(*
version 1.0	4 aug 2006
programmer 	hugo
tested by		tobias

this Function Block extracts the 8 Bits from a byte

executioin TIME on wago 750-841 = 13us
*)
B0 := IN.0;
B1 := IN.1;
B2 := IN.2;
B3 := IN.3;
B4 := IN.4;
B5 := IN.5;
B6 := IN.6;
B7 := IN.7;
END_FUNCTION_BLOCK

(* POU Engineering/signal processing/Byte_to_Range, ST *)
FUNCTION Byte_to_Range : REAL
VAR_INPUT
	X : BYTE;
	low : REAL;
	high : REAL;
END_VAR
VAR
END_VAR

(*
version 1.0	9. jan 2008
programmer 	hugo
tested by		tobias

Byte_to_Range converts a Byte into a real between low and high.

*)
Byte_to_Range := (high - low) * X / 255.0 + low;


(* revision history
hm	9. jan 2008		rev 1.0
	original version

*)
END_FUNCTION

(* POU String/BYTE_TO_STRH, ST *)
FUNCTION BYTE_TO_STRH : STRING
VAR_INPUT
	IN : BYTE;
END_VAR
VAR
	temp : BYTE;
	PT : POINTER TO BYTE;
END_VAR

(*
version 1.2	15 dec 2007
programmer 	hugo
tested by		tobias

BYTE_TO_STRINGH converts a Byte to a String of Hexadecimal represented by '0' .. '9' and 'A' .. 'F'.
The lowest order Character will be on the right and the high order Character on the left.

*)
(* read pointer to output string *)
PT := ADR(BYTE_TO_STRH);
(* calculate high order hex value *)
temp := SHR(in,4);
(* convert value to hex character *)
IF temp <= 9 THEN temp := temp + 48; ELSE temp := temp + 55; END_IF;
(* write friat character to output string *)
PT^ := temp;
(* calculate low order hex value *)
temp := in AND 2#00001111;
IF temp <= 9 THEN temp := temp + 48; ELSE temp := temp + 55; END_IF;
(* increment pointer and wirte low order character *)
pt := pt + 1;
pt^ := temp;
(* set pointer at the end of the output string and close the string with 0 *)
pt := pt + 1;
pt^:= 0;


(* code before rev 1.2
FOR i := 1 TO 2 DO
	X := in AND 2#1111;
	IF X <= 9 THEN X := X + 48; ELSE X := X + 55; END_IF;
	Cx := CHR(X);
	temp := CONCAT(Cx, temp);
	in := SHR(in,4);
END_FOR;
BYTE_TO_STRH := temp;
*)

(* revision history

hm		9.6.2007		rev 1.0		
	original version 

hm		11.9.2007		rev 1.1		
	changed coding for compatibility with twincat, under twincat concat cannot have a function as argument.	

hm		15 dec 2007		REV 1.2
	changed code for higher performance
*)
END_FUNCTION

(* POU Engineering/conversion/C_to_F, ST *)
FUNCTION C_to_F : REAL
VAR_INPUT
	celsius : REAL;
END_VAR
VAR
END_VAR

(*
version 1.0	4 aug 2006
programmer 	hugo
tested by		tobias

this function converts celsius  to fahrenheit 

*)
C_to_F := celsius * 1.8 + 32;
END_FUNCTION

(* POU Engineering/conversion/C_to_K, ST *)
FUNCTION C_to_K : REAL
VAR_INPUT
	Celsius : REAL;
END_VAR
VAR
END_VAR

(*
version 1.0	4 dec 2006
programmer 	hugo
tested by		tobias

this function converts celsius to kelvin
*)
C_to_K := Celsius - 273.15;
END_FUNCTION

(* POU Mathematical/Complex/CABS, ST *)
FUNCTION CABS : REAL
VAR_INPUT
	X : complex;
END_VAR
VAR
END_VAR

(*
version 1.0	21 feb 2008
programmer 	hugo
tested by	oscat

this function the aboslute value of a complex number

*)
CABS := HYPOT(x.re, x.im);


(* revision history
hm	21. feb 2008	rev 1.0
	original version

*)
END_FUNCTION

(* POU Engineering/measurements/Calibrate, ST *)
FUNCTION_BLOCK Calibrate
VAR_INPUT
	X : REAL;
	CO : BOOL;
	CS : BOOL;
END_VAR
VAR_INPUT CONSTANT
	Y_Offset : REAL;
	Y_Scale : REAL;
END_VAR
VAR_OUTPUT
	Y : REAL;
END_VAR
VAR RETAIN
	offset : REAL;
	Scale : REAL := 1;
END_VAR

(*
	version 1.2	22 feb 2007
	programmer 	hugo
	tested BY		hans

Calibrate allows for offset and scale calibration of an analog input.
offset is calibrated to a stored reference Y_offset while CO is true.
after the offset is calibrated, scale can be calibrated to a reference value Y_scale while CS is true.
*)
(* check for calibration *)
IF CO THEN
	Offset := Y_Offset - X;
ELSIF CS THEN
	scale := Y_scale / (X+Offset);
END_IF;
(* calculate output *)
Y := (X + Offset) * Scale;


(* revision history
hm 22.2.2007		rev 1.2
	changed VAR RETAIN PERSISTENT to VAR RETAIN for better compatibility
	wago lon contollers do not support persisitent

*)
END_FUNCTION_BLOCK

(* POU String/CAPITALIZE, ST *)
FUNCTION CAPITALIZE : STRING
VAR_INPUT
	str : STRING;
END_VAR
VAR
	PT : POINTER TO BYTE;
	pos : INT;
	L : INT;
	first : BOOL := TRUE;
END_VAR

(*
version 1.0	4. mar 2008
programmer 	hugo
tested by		tobias

uppercase returns str while all letters a..z and ä,ö,ü are converted to uppercase

*)
PT := ADR(CAPITALIZE);
CAPITALIZE := str;
L := LEN(str);
FOR pos := 1 TO l DO
	IF first THEN
		pt^ := TO_UPPER(pt^);
	END_IF;
	(* remember in first if the next char needs to capitalized *)
	IF pt^ = 32 THEN first := TRUE; ELSE first := FALSE; END_IF;
	PT := pt + 1;
END_FOR;

(* revision histroy
hm		4. mar 2008	rev 1.0
	original release

*)	
END_FUNCTION

(* POU String/TO_UPPER, ST *)
FUNCTION TO_UPPER : BYTE
VAR_INPUT
	IN : BYTE;
END_VAR
VAR
END_VAR

(*
version 1.0	6 mar 2008
programmer 	hugo
tested by		tobias

to_upper converts a character from lowercase to uppercase

*)
IF extended_ascii THEN
	IF ((in > 96) AND (in < 123)) OR ((in > 223) AND (in <> 247) AND (in <> 255)) THEN
		TO_UPPER := in AND 16#DF;
	ELSE
		TO_UPPER := in;
	END_IF;
ELSE
	IF ((in > 96) AND (in < 123)) THEN
		TO_UPPER := in AND 16#DF;
	ELSE
		TO_UPPER := in;
	END_IF;
END_IF;

(* revision history
hm		6. mar 2008	rev 1.0
	original version

*)
END_FUNCTION

(* POU Mathematical/Complex/CARG, ST *)
FUNCTION CARG : REAL
VAR_INPUT
	X : complex;
END_VAR
VAR
END_VAR

(*
version 1.0	21 feb 2008
programmer 	hugo
tested by	oscat

this function calculates the phase angle (argument) of a complex number

*)
CARG := ATAN(X.im / X.re);



(* revision history
hm	21. feb 2008	rev 1.0
	original version


*)
END_FUNCTION

(* POU Mathematical/Complex/CCON, ST *)
FUNCTION CCON : complex
VAR_INPUT
	X : complex;
END_VAR
VAR
END_VAR

(*
version 1.0	21 feb 2008
programmer 	hugo
tested by	oscat

this function calcucates the conjugation of a complex number

*)
CCON.re := x.re;
CCON.im := -x.im;


(* revision history
hm	21. feb 2008	rev 1.0
	original version

*)
END_FUNCTION

(* POU Logic/gate logic/check_parity, ST *)
FUNCTION check_parity : BOOL
VAR_INPUT
	in : DWORD;
	p : BOOL;
END_VAR
VAR
END_VAR

(*
version 1.3	18 feb 2008
programmer 	hugo
tested by		tobias

this function checks for an even partity for a dword and partity bit.

*)
check_parity := NOT p;
WHILE in > 0 DO
	check_parity := check_parity XOR in.0 XOR in.1 XOR in.2 XOR in.3;
	in := SHR(in,4);
END_WHILE;

(* code before rev 1.2
WHILE in > 0 DO
	IF in.0 THEN cnt := cnt + 1; END_IF;
	in := SHR(in,1);
END_WHILE;
check_parity := even(cnt) XOR P;
*)


(* revision history

rev 1.0 HM  1.oct.2006

rev 1.1 hm	10.sep.2007
	changed algorithm to improove performance

rev 1.2	hm	8 dec 2007
	changed algorithm to improove performance

rev 1.3 hm	18. feb 2008
	changed algorithm to improove performance
*)
END_FUNCTION

(* POU String/CHR, ST *)
FUNCTION CHR : STRING
VAR_INPUT
	C : BYTE;
END_VAR
VAR
	PT : POINTER TO BYTE;
END_VAR

(*
version 1.1	4. feb 2008
programmer 	hugo
tested by		tobias

CHR creates a character from a byte input and stuffs it in a one character length string.

*)
PT := ADR(CHR);
PT^ := C;
pt := pt + 1;
pt^ := 0;

(* revision history
hm		16 jan 2007		rev 1.0
	original version

hm		4. feb. 2008		rev 1.1
	return string would not be terminated properly
*)
END_FUNCTION

(* POU Mathematical/Geometry/circle_A, ST *)
FUNCTION circle_A : REAL
VAR_INPUT
	rx : REAL;
	ax : REAL;
END_VAR
VAR
END_VAR

(*
version 1.2	22. feb 2008
programmer 	hugo
tested by		tobias

circle_A calculates the Area of a circle segement if ax = 360 the whole circle is calculated


*)
circle_A := Rx * RX * 8.726646E-3 * Ax;

(* revision histroy
hm	16. oct 2007	rev 1.0
	original version

hm	4. dec 2007		rev 1.1
	changed code for better performance

hm	22. feb 2008	rev 1.2
	improved performance
*)
END_FUNCTION

(* POU Mathematical/Geometry/circle_C, ST *)
FUNCTION circle_C : REAL
VAR_INPUT
	Rx : REAL;
	Ax : REAL;
END_VAR
VAR
END_VAR

(*
version 1.1	22 feb 2008
programmer 	hugo
tested by		tobias

circle_C calculates the Circumference of a circle  if ax = 360 the whole circle is calculated

*)
circle_C := 1.7453293E-2 * Rx * Ax;

(* revision histroy
hm	16. oct 2007	rev 1.0
	original version

hm	22. feb 2008	rev 1.1
	improved performance
*)
END_FUNCTION

(* POU Building/electrical/click, ST *)
FUNCTION_BLOCK click
VAR_INPUT
	in : BOOL;
END_VAR
VAR_OUTPUT
	Q : BOOL;
	single : BOOL;
	double : BOOL;
	triple : BOOL;
	status: BYTE;
END_VAR
VAR_INPUT CONSTANT
	T_debounce : TIME := t#10ms;
	T_short : TIME := t#200ms;
	T_pause : TIME := t#500ms;
	T_reconfig : TIME := t#1m;
END_VAR
VAR
	debounce : TON;
	tx : TIME;
	last : TIME;
	init : BOOL;
	edge : BOOL;
	standby: BOOL;
	state: INT;
END_VAR

(*
version 1.2	15 sep 2007
programmer 	oscat
tested by		tobias

click checks an input for single, double or tripple click and sets the corresponding output single, doulbe or triple for the time the input stays high at the last click.
the maximum high and low time for a click can beconfigrured with setup variables.
the input cinfigures itself to be high or low active dependung on which state the input stays longer than t_reconfig.

*)
(* read system time *)
tx := DWORD_TO_TIME(T_PLC_MS());

(* set last and tx if never started before *)
IF NOT init THEN
	init := TRUE;
	last := tx;
	debounce.PT := T_debounce;
	standby := in;
END_IF;

(* debounce input *)
debounce(in := in XOR standby);
Q := debounce.Q;

(* delete outputs if input is inactive *)
IF NOT Q THEN
	single := FALSE;
	double := FALSE;
	triple := FALSE;
	status := 110;
END_IF;

(* check for input edge *)
IF Q XOR edge THEN
	edge := in;
	last := tx;
	IF Q THEN state := state + 1; END_IF;
END_IF;

IF (q AND tx - last >= T_short) OR (NOT q AND tx - last >= t_pause) THEN
	CASE state OF
		1:	single := TRUE;
			status := 111;
		2:	double := TRUE;
			status := 112;
		3:	triple := TRUE;
			status := 113;
	END_CASE;
	state := 0;
END_IF;

(* determine if high or low active *)
IF tx - last >= t_reconfig THEN
	standby := in;
	last := tx;
END_IF;



(* revision history

15 Feb 2007	rev 1.0	hm
	created original version

18.5.2007		rev 1.1 hm
	corrected an error while execution would stop after t_reconfig elapsed.

15.9.2007		rev 1.2 hm
	replaced Time() with T_PLC_MS for compatibility and performance reasons

*)
END_FUNCTION_BLOCK

(* POU Logic/generators/clk_div, ST *)
FUNCTION_BLOCK clk_div
VAR_INPUT
	clk : BOOL;
	rst: BOOL;
END_VAR
VAR_OUTPUT
	Q0 : BOOL := 0;
	Q1 : BOOL := 0;
	Q2 : BOOL := 0;
	Q3 : BOOL := 0;
	Q4 : BOOL := 0;
	Q5 : BOOL := 0;
	Q6 : BOOL := 0;
	Q7 : BOOL := 0;
END_VAR
VAR
	cnt: BYTE := 0;
END_VAR

(*
version 1.1	2 jan 2008
programmer 	hugo
tested by		tobias

this is a clock divider
each output divides the signal by 2
Q0 = clk / 2 , Q1 = Q0 / 2 and so on.
the outputs have a 50% duty cycle each.


*)
IF rst THEN
	cnt:= 0;
	Q0 := 0;
	Q1 := 0;
	Q2 := 0;
	Q3 := 0;
	Q4 := 0;
	Q5 := 0;
	Q6 := 0;
	Q7 := 0;
ELSIF clk THEN
	cnt:= cnt +1;
	Q0 := cnt.0;
	Q1 := cnt.1;
	Q2 := cnt.2;
	Q3 := cnt.3;
	Q4 := cnt.4;
	Q5 := cnt.5;
	Q6 := cnt.6;
	Q7 := cnt.7;
END_IF;

(* revision history
hm	4. aug. 2006	rev 1.0
	original version

hm	2. jan 2008		rev 1.1
	improved performance

*)
END_FUNCTION_BLOCK

(* POU Logic/generators/CLK_N, ST *)
FUNCTION_BLOCK CLK_N
VAR_INPUT
	N : INT;
END_VAR
VAR_OUTPUT
	Q : BOOL;
END_VAR
VAR
	edge : BOOL := 0;
	stime: DWORD;
	clk: BOOL;
END_VAR

(*
version 1.0	17 sep 2007
programmer 	hugo
tested by		tobias

clk_N uses the internal sps time to generate one pulse every N ms
every pulse is only valid for one cycle so that a edge trigger is not necessary
clk_N generates pulses depending on the accuracy of the system clock.
The input N controlls the period time of the clock.
N=0 equals 1ms, N=1 equals 2ms, N=2 equals 4ms, N=3 equals 8ms ....

be careful, 1ms clocks will only work on very powerful sps cpu's
*)
stime := SHR(T_PLC_MS(),N);
clk := stime.0;
Q := clk XOR edge;
edge := CLK;

(* revision history
hm	16. dec 2007		rev 1.0
	original version

*)
END_FUNCTION_BLOCK

(* POU XTEST/Ideas/stime, ST *)
FUNCTION_BLOCK stime
VAR_INPUT
END_VAR
VAR_OUTPUT
	tx : DWORD;
END_VAR
VAR
	last_time: DWORD;
	bit31: BOOL;
END_VAR

(* this function block makes sure that the timer of a siemens sps counts from 0 - 2^32-1. *)
(* this FB is only necessary for siemens sps
the siemens sps timer counts from 0 to 2^31-1 and starts at 0 sfter overrun.
this means that the bit 31 (the highest bit ) will never be used and therefore
a problem arises when t2 - t1 is checked.
t2 - t1 is always valid also in an timer overrun situation where the time t1 is very high and t2 is very low.
the result of the subtraction t2 - t1 however is still valid.
this calculation does not work for siemens because the highest bit is not used.

this module stores the highest bit, changes the highest bit at every overrun occurence and stuffs ther highest bit in the output.
the output is then used by t_plc_us and t_plc_ms.

the correction needs and fb and not a function because the value of the highest bit has to be stored.

do never use this function block in a codesys environment. the timer in codesys is correct and runs from 0 to 2^32-1
*)

(* read the system timer *)
tx := TIME_TO_DWORD(TIME());

(* check for overrun *)
IF tx < last_time THEN
	(* an overrun has occured, change the value of the highest bit *)
	bit31 := NOT bit31;
END_IF;

(* remember the last system time for the next overrun check *)
last_time := tx;

(* stuff the highest bit into the timer value *)
tx.31 := bit31;
END_FUNCTION_BLOCK

(* POU Logic/generators/CLK_Prg, ST *)
	FUNCTION_BLOCK CLK_Prg
VAR_INPUT
	PT : TIME := t#10ms;
END_VAR
VAR_OUTPUT
	Q : BOOL := 0;
END_VAR
VAR
	init : BOOL := FALSE;
	last : TIME;
	tx: TIME;
END_VAR

(*
version 1.2	17 sep 2007
programmer 	hugo
tested by		tobias

clk_prg uses the internal sps time to generate a clock with programmable period time.
the period time is defined for 10ms .. 65s
the first cycle after start is a clk pulse and then depending on the programmed period time a delay.
every pulse is only valid for one cycle.
the accuracy of clk_prg is depending on the accuracy of the system clock.

*)
(* read system time *)
tx := DWORD_TO_TIME(T_PLC_MS());

(* initialize on startup *)
IF NOT init THEN
	init := TRUE;
	last := tx - pt;
END_IF;

(* generate output pulse when next_pulse is reached *)
IF tx - last >= pt THEN
	Q := TRUE;
	last := tx;
ELSE
	Q := FALSE;
END_IF;


(* revision hiostory

hm 25 feb 2007	rev 1.1
	rewritten code for higher performance
	pt can now be changed during runtime

hm	17. sep 2007	rev 1.2
	replaced time() with t_plc_ms() for compatibility reasons

*)
END_FUNCTION_BLOCK

(* POU Logic/generators/CLK_Pulse, ST *)
FUNCTION_BLOCK CLK_Pulse
VAR_INPUT
	PT : TIME := t#10ms;
	N : INT := 0;
	rst : BOOL := 0;
END_VAR
VAR_OUTPUT
	Q : BOOL := 0;
	cnt : INT := 0;
	run : BOOL := 0;
END_VAR
VAR
	pti : TIME := t#0ms;
	next_pulse: TIME := T#0s;
	overflow: BOOL := FALSE;
	tx: TIME;
END_VAR

(*
version 1.1	17 sep 2007
programmer 	hugo
tested by		tobias

clk_pulse uses the internal sps time to generate a clock with programmable period time.
the period time is defined for 10ms .. 65s.
pulse generation is continuous if N = 0 and for n pulses otherwise.
if the period time is set to less then 10ms the min clock perid is 10ms.
the first cycle after start is a clk pulse and then depending on the programmed period time a delay.
every pulse is only valid for one cycle so that a edge trigger is not necessary
clk_prg depending on the accuracy of the system clock.

*)
(* read system *)
tx := DWORD_TO_TIME(T_PLC_MS());


IF rst THEN
	run := FALSE;
	pti := t#0ms;
	next_pulse := t#0ms;
	overflow := FALSE;
	Q := FALSE;
	cnt := 0;
ELSIF cnt <= N OR N = 0 THEN
	IF NOT run THEN
		next_pulse := tx;
		run := TRUE;
		IF pt < T#10ms THEN PTI := T#10ms; ELSE pti := pt; END_IF;
	END_IF;
	IF tx >= next_pulse AND NOT overflow AND (cnt < N OR N = 0) THEN
		Q := TRUE;
		cnt := cnt + 1;
		IF next_pulse + pti < next_pulse THEN
			overflow := TRUE;
		END_IF;
		next_pulse := next_pulse + pti;
	ELSE
		Q := FALSE;
		IF cnt = N THEN run := FALSE; END_IF
		IF tx <= next_pulse THEN overflow := FALSE; END_IF;
	END_IF;
END_IF

(* revision history
hm		4. aug 2006		rev 1.0
	original version

hm		17. sep 2007	rev 1.1
	replaced time() with T_PLC_S() fr compatblity reasons

*)
END_FUNCTION_BLOCK

(* POU Mathematical/Geometry/cone_V, ST *)
FUNCTION cone_V : REAL
VAR_INPUT
	rx : REAL;
	hx : REAL;
END_VAR
VAR
END_VAR

(*
version 1.1	4 dec 2007
programmer 	hugo
tested by		tobias

cone_V calculates the Volume of a cone

*)
cone_V := 1.047197551 * RX * RX * hx;

(* revision histroy
hm	17. oct 2007	rev 1.0
	original version

hm	4. dec 2007		rev 1.1
	changed code for better performance

hm	22. feb 2008	rev 1.2
	changed code for better performance
*)
END_FUNCTION

(* POU Engineering/control/control_set1, ST *)
FUNCTION_BLOCK control_set1
VAR_INPUT
	Kt : REAL;
	Tt : REAL;
	PI : BOOL;
	PID : BOOL;
END_VAR
VAR_INPUT CONSTANT
	P_K : REAL := 0.5;
	PI_K : REAL := 0.45;
	PI_TN : REAL := 0.83;
	PID_K : REAL := 0.6;
	PID_TN : REAL := 0.5;
	PID_TV : REAL := 0.125;
END_VAR
VAR_OUTPUT
	KP : REAL;
	TN : REAL;
	TV : REAL;
	KI : REAL;
	KD : REAL;
END_VAR
VAR
END_VAR

(*
version 1.0	4 nov 2007
programmer 	hugo
tested by	tobias

takahashi calculates controller parameters for P, PI and PID controllers based on the ziegler nichols method.

*)
IF pi AND PID THEN
	KP := 0;
	TN := 0;
	TV := 0;
ELSIF PID THEN
	KP := PID_K * Kt;
	TN := PID_TN * Tt;
	TV := PID_TV * Tt;
ELSIF PI THEN
	KP := PI_K * Kt;
	TN := PI_TN * Tt;
ELSE
	KP := P_K * Kt;
END_IF;

(* KI and KD are calculated *)
IF tn > 0 THEN KI := KP / TN; ELSE KI := 0; END_IF;
KD := KP * TV;

(* revision history
hm	4. nov 2007		rev 1.0
	original version

*)
END_FUNCTION_BLOCK

(* POU Engineering/control/control_set2, ST *)
FUNCTION_BLOCK control_set2
VAR_INPUT
	KS : REAL;
	TU : REAL;
	TG : REAL;
	PI : BOOL;
	PID : BOOL;
END_VAR
VAR_INPUT CONSTANT
	P_K : REAL := 1.0;
	PI_K : REAL := 0.9;
	PI_TN : REAL := 3.33;
	PID_K : REAL := 1.2;
	PID_TN : REAL := 2;
	PID_TV : REAL := 0.5;
END_VAR
VAR_OUTPUT
	KP : REAL;
	TN : REAL;
	TV : REAL;
	KI : REAL;
	KD : REAL;
END_VAR
VAR
	TX : REAL;
END_VAR

(*
version 1.0	4 nov 2007
programmer 	hugo
tested by	tobias

takahashi calculates controller parameters for P, PI and PID controllers based on the ziegler nichols method.

*)
IF TU > 0 AND KS > 0 THEN TX := TG/TU/KS; END_IF;
IF pi AND PID THEN
	KP := 0;
	TN := 0;
	TV := 0;
ELSIF PID THEN
	KP := PID_K * TX;
	TN := PID_TN * TU;
	TV := PID_TV * TU;
ELSIF PI THEN
	KP := PI_K * TX;
	TN := PI_TN * TU;
ELSE
	KP := P_K * TX;
END_IF;

(* KI and KD are calculated *)
IF TN > 0 THEN KI := KP / TN; ELSE KI := 0; END_IF;
KD := KP * TV;

(* revision history
hm	4. nov 2007		rev 1.0
	original version

*)
END_FUNCTION_BLOCK

(* POU Logic/FF edge triggered/COUNT_BR, ST *)
FUNCTION_BLOCK COUNT_BR
VAR_INPUT
	SET : BOOL;
	IN : BYTE;
	UP : BOOL;
	DN : BOOL;
	STEP : BYTE := 1;
	MX : BYTE := 255;
	RST : BOOL;
END_VAR
VAR_INPUT CONSTANT

END_VAR
VAR_OUTPUT
	CNT : BYTE;
END_VAR
VAR
	last_up: BOOL;
	last_dn: BOOL;
END_VAR

(*
	version 1.0	16 jan 2008
	programmer 	hugo
	tested BY	tobias

Count_R is a byte counter with independen up and dn inputs. the counter counts from 0 to mx and continues at 0 after is has reached mx
a step input sets the counters stepping width.

*)
IF rst THEN
	cnt := 0;
ELSIF set THEN
	cnt := LIMIT(0,in,mx);
ELSIF up AND NOT last_up THEN
	cnt := INT_TO_BYTE(inc(cnt,step,mx));
ELSIF dn AND NOT last_dn THEN
	cnt := INT_TO_BYTE(inc(cnt,-step,mx));
END_IF;
last_up := up;
last_dn := dn;

(* revision history
hm	16. jan 2008	rev 1.0
	original version

*)
END_FUNCTION_BLOCK

(* POU String/COUNT_CHAR, ST *)
FUNCTION COUNT_CHAR : INT
VAR_INPUT
	str : STRING;
	chr : BYTE;
END_VAR
VAR
	l: INT;
	pt : POINTER TO BYTE;
	pos: INT;
END_VAR


(*
version 1.0	29. feb 2008
programmer 		kurt
tested by		hugo

COUNT_CHAR how often a character CHAR occurs within a string STR.

*)
PT := ADR(str);
l := LEN(str);
COUNT_CHAR := 0;
FOR pos := 1 TO l DO
	IF pt^ = CHR THEN COUNT_CHAR := COUNT_CHAR + 1; END_IF;
    PT := PT + 1;
END_FOR;


(* revision history
hm		29. feb 2008	rev 1.0
	original version

*)
END_FUNCTION

(* POU Mathematical/Complex/CPOL, ST *)
FUNCTION CPOL : complex
VAR_INPUT
	L : REAL;
	A : REAL;
END_VAR
VAR
END_VAR

(*
version 1.0	21 feb 2008
programmer 	hugo
tested by	oscat

this function creates a complex numbers for the polar form with the inputs L (length) an A for Angle.

*)
CPOL.re := L * COS(A);
CPOL.im := L * SIN(A);


(* revision history
hm	21. feb 2008	rev 1.0
	original version

*)
END_FUNCTION

(* POU Logic/Others/CRC_CHECK, ST *)
FUNCTION CRC_CHECK : BOOL
VAR_INPUT
	pt : POINTER TO ARRAY[0..32000] OF BYTE;
	size : INT;
END_VAR
VAR_INPUT CONSTANT
	Polynom_L : DWORD;
	Polynom_32 : BOOL;
END_VAR
VAR
	temp: DWORD;
END_VAR

(*
version 1.0	9 jun 2007
programmer 	hugo
tested by		tobias

CRC_CHECK checks a block of data for a crc checksum and returns true is the checksum is 0 and therfore a error free data transmission.
the CRC Polynom is specified with the config variable Polynom_L which holds the lowest 32 bits of the polynom and Polynom_33 which holds bit 33 of the Polynom.
A Polynom x4 + X + 1 is represented by 10011.
The input data is an array of byte of any size, the function is called by CRC_CHECK(ADR(array),SIZEOF(array)).

*)
temp := CRC_GEN(pt, size, polynom_L, polynom_32, 0, 0, FALSE, FALSE);
IF temp = 0 THEN CRC_CHECK := TRUE; ELSE CRC_CHECK := FALSE; END_IF;

(* typical crc polynoms

CRC-4-ITU 			x4 + x + 1 					(ITU G.704, p. 12) 	0x3 or 0xC (0x9)
CRC-5-ITU 			x5 + x4 + x2 + 1 			(ITU G.704, p. 9) 	0x15 or 0x15 (0x0B)
CRC-5-USB 			x5 + x2 + 1 				(use: USB token packets) 	0x05 or 0x14 (0x9)
CRC-6-ITU 			x6 + x + 1 					(ITU G.704, p. 3) 	0x03 or 0x30 (0x21)
CRC-7 				x7 + x3 + 1 				(use: telecom systems, MMC) 	0x09 or 0x48 (0x11)
CRC-8-ATM 			x8 + x2 + x + 1 				(use: ATM HEC) 	0x07 or 0xE0 (0xC1)
CRC-8-CCITT 		x8 + x7 + x3 + x2 + 1 		(use: 1-Wire bus) 	0x8D or 0xB1 (0x63)
CRC-8-Dallas/Maxim 	x8 + x5 + x4 + 1 			(use: 1-Wire bus) 	0x31 or 0x8C (0x19)
CRC-8 				x8 + x7 + x6 + x4 + x2 + 1 	0xD5 or 0xAB (0x57)
CRC-8-SAE J1850 	x8 + x4 + x3 + x2 + 1 		0x1D or 0xB8
CRC-10 				x10 + x9 + x5 + x4 + x + 1 	0x233 or 0x331 (0x263)
CRC-12 				x12 + x11 + x3 + x2 + x + 1 (use: telecom systems) 	0x80F or 0xF01 (0xE03)
CRC-15-CAN 			x15 + x14 + x10 + x8 + x7 + x4 + x3 + 1 	0x4599 or 0x4CD1 (0x19A3)
CRC-16-Fletcher 	Not a CRC; see Fletcher's checksum 	Used in Adler-32 A & B CRCs
CRC-16-CCITT 	x16 + x12 + x5 + 1 (XMODEM,X.25, V.41, Bluetooth, PPP, IrDA; known as "CRC-CCITT") 	0x1021 or 0x8408 (0x0811)
CRC-16-IBM 	x16 + x15 + x2 + 1 (USB, many others; also known as "CRC-16") 	0x8005 or 0xA001 (0x4003)
CRC-24-Radix-64 	x24 + x23 + x18 + x17 + x14 + x11 + x10 + x7 + x6 + x5 + x4 + x3 + x + 1 	0x864CFB or 0xDF3261 (0xBE64C3)
CRC-32-Adler 	Not a CRC; see Adler-32 	See Adler-32
CRC-32-MPEG2 	x32 + x26 + x23 + x22 + x16 + x12 + x11 + x10 + x8 + x7 + x5 + x4 + x2 + x + 1 	0x04C11DB7 or 0xEDB88320 (0xDB710641) Also used in IEEE 802.3
CRC-32-IEEE 802.3 	x32 + x26 + x23 + x22 + x16 + x12 + x11 + x10 + x8 + x7 + x5 + x4 + x2 + x + 1 (V.42) 	0x04C11DB7 or 0xEDB88320 (0xDB710641)
CRC-32C (Castagnoli) 	x32 + x28 + x27 + x26 + x25 + x23 + x22 + x20 + x19 + x18 + x14 + x13 + x11 + x10 + x9 + x8 + x6 + 1 	0x1EDC6F41 or 0x82F63B78 (0x05EC76F1)
CRC-64-ISO 	x64 + x4 + x3 + x + 1 (use: ISO 3309) 	0x000000000000001B or 0xD800000000000000 (0xB000000000000001)
CRC-64-ECMA-182 	x64 + x62 + x57 + x55 + x54 + x53 + x52 + x47 + x46 + x45 + x40 + x39 + x38 + x37 + x35 + x33 + x32 + x31 + x29 + x27 + x24 + x23 + x22 + x21 + x19 + x17 + x13 + x12 + x10 + x9 + x7 + x4 + x + 1
(as described in ECMA-182 p.63) 	0x42F0E1EBA9EA3693 or 0xC96C5795D7870F42 (0x92D8AF2BAF0E1E85)

*)

(* revision history

hm		9.6.2007	rev 1.0		original version 

*)
END_FUNCTION

(* POU Logic/generators/D_Trig, ST *)
FUNCTION_BLOCK D_Trig
VAR_INPUT
	in : DWORD;
END_VAR
VAR_OUTPUT
	Q : BOOL;
	X : DWORD;
END_VAR
VAR
	last_in : DWORD;
END_VAR

(*
version 1.1	19. feb 2008
programmer 	hugo
tested by		tobias

this block is similar to the IEC Standard R_trig and F_trig but it monitors a DWORD, WORD or Byte Variable instead and generated an Output Pulse for one cycle only when the input has changed.
an additional output x (Dword) will state the chage of the input.
Example: the input has chaged from 0001 to 0010 then the output x will be 2.

*)
Q := in <> last_in;
X := in - last_in;
last_in := in;


(* revision history

hm 	4.09.2007		rev 1.0
	original version released

hm	19. feb. 2008	rev 1.1
	performance improvement
*)
END_FUNCTION_BLOCK

(* POU XTEST/Baustein Tests/date_test, ST *)
FUNCTION_BLOCK date_test
VAR_INPUT
END_VAR
VAR_OUTPUT
	fail : STRING;
	error : BOOL := FALSE;
	jahr : INT;
END_VAR
VAR
	i: INT;
	test : DATE;
	jan1 : DATE;
	dez31 : DATE;
END_VAR
IF error THEN RETURN; END_IF;

FOR i := 1970 TO 2099 DO
	jan1 := set_Date(i,1,1);
	dez31 := set_Date(i,12,31);

	(* test der funktion year_begin *)
	test := year_begin(i);
	IF test <> jan1 THEN
		error := TRUE;
		jahr := i;
		FAIL := 'year_begin';
	END_IF;

	(* test year *)
	IF year(jan1) <> i OR year(dez31) <> i THEN
		error := TRUE;
		jahr := i;
		fail := 'year';
	END_IF;
END_FOR;
END_FUNCTION_BLOCK

(* POU Time&Date/day_of_date, ST *)
FUNCTION day_of_date : INT
VAR_INPUT
	idate : DATE;
END_VAR
VAR
END_VAR


(*
	version 1.1	1 okt 2007
	programmer 	oscat
	tested BY		oscat

DAY_OF_DATE returns the days since 1.1.1970

*)
IF STEP7 THEN
	(* adjust step7 day by 7305 days because step7 date fornat starts at 1.1.1990  *)
	day_of_date := DWORD_TO_INT(DATE_TO_DWORD(idate) / 86400) + 7305;
ELSE
	day_of_date := DWORD_TO_INT(DATE_TO_DWORD(idate) / 86400);
END_IF;


(* revision history
hm		16.9.2007		rev 1.0
	original version

hm		1. okt 2007		rev 1.1
	added step7 compatibility

*)
END_FUNCTION

(* POU Time&Date/day_to_time, ST *)
FUNCTION day_to_time : TIME
VAR_INPUT
	input : REAL;
END_VAR
VAR
END_VAR

(*
version 1.0	4 aug 2006
programmer 	hugo
tested by		tobias

converts an amount of days in real to time 
*)
day_to_time := DWORD_TO_TIME(REAL_TO_DWORD(input * 86400000));
END_FUNCTION

(* POU Time&Date/days_delta, ST *)
FUNCTION days_delta : INT
VAR_INPUT
	date_1 : DATE;
	date_2 : DATE;
END_VAR
VAR
END_VAR

(*
version 1.1	27 dec 2006
programmer 	hugo
tested by		tobias

days_delta calculates the days between two dates. the days are calculated date_2 - date_1.

*)
days_delta := day_of_date(date_2) - day_of_date(date_1);

(* revision history
hm	27. dec 2006	rev 1.0
	original version

hm	16.9.2007		rev 1.1
	coorected an error in formula and changed algorithm to show positive and negative delta

*)
END_FUNCTION

(* POU Time&Date/DCF77, ST *)
FUNCTION_BLOCK DCF77
VAR_INPUT
	rec : BOOL;
	sdt : DT;
END_VAR
VAR_INPUT CONSTANT
	sync_timeout : TIME := t#2m;
	time_offset : INT := 1;
	dst_en : BOOL := TRUE;
END_VAR
VAR_OUTPUT
	TP : BOOL;
	DST : BOOL;
	weekday : INT;
	error: BOOL := TRUE;
	RTC : DT;
	RTC1 : DT;
	msec : INT;
	sync : BOOL;
END_VAR
VAR
	MEZ : DT;
	UTC : DT;
	state : INT;
	edge: BOOL;
	tx : TIME;
	ty: TIME;
	last : TIME;
	bits : ARRAY[0..58] OF BOOL;
	cnt : INT;
	i : INT;
	old_time : DT;
	minute : INT;
	hour : INT;
	day : INT;
	month : INT;
	year : INT;
	last_sync: TIME;
	t1: TIME;
	tz: TIME;
	init: BOOL;
END_VAR


(*
version 1.7	23. jan 2008
programmer 	hugo
tested by		tobias

this is a decoder for a DCF77 signal.
the decoder decodes the DCF77 signal and checks for a valid Date_Time.
since the dcf77 signal is only secured with a simple parity the decoder waits for two consecutive valid transmissions before it sets the output signals.
given a valid reception by the receiver the decoder can take up to 3 minutes to start its clocks the first time.
after a valid signal is detected the error output goes low and dignals a valid dcf signal from the receiver.
a tp is only valid for one program cycle to allow for external rtc setting.
after a valid signal is detected two independent internal clocks are started (RTC and RTC1), the seconds  of these clocks are generated by software since the dcf signal is only valid for minutes.
rtc is always utc ( world time) and rtc1 can be set to any time zone by setting the time_zone_offset and enabling dst for automatic summertime.
a sync output signals the the rtc and rtc1 are in sync with the dcf77 signal, if the dcf77 signal is lost for more then the sync time the sync output goes low
but the rtc and rtc1 outputs keep running based on software timing until a valid dcf77 signal is received again and triggers the clock.
in addition a millisecond output gives further resolutionof the clocks.
a dst output shows if daylight saving time is enables and the weekday output shows which day of week currently is ( 1= monday ... 7= sunday).


*)
(* if tp was set it should only be active for 1 cycle *)
TP := FALSE;

(* read system time *)
t1 := DWORD_TO_TIME(T_PLC_MS());
tx := t1 - last;

IF rec XOR edge THEN
	edge := rec;
	IF NOT rec AND tx > t#1700ms AND tx < t#2000ms THEN
		(* start condition reached *)
		state := 0;
		tp := NOT error;
	ELSIF NOT rec AND tx > t#700ms AND tx < t#1000ms THEN
		(* second switch detected *)
		IF state < 58 THEN state := state +1; ELSE state := 0; END_IF;
	ELSIF rec AND tx  < t#120ms THEN
		(* bit 0 detected  *)
		bits[state] := 0;
	ELSIF rec AND tx > t#120ms AND tx < t#250ms THEN
		(* bit 1 detected *)
		bits[state] := 1;
	ELSE
		(* error condition received signal is not valid *)
		error := TRUE;
		state := 0;
	END_IF;
	last := last + tx;
	IF rec AND state = 58 THEN
		error := FALSE;

		(* decode the bits and check for possible errors *)
		IF bits[0] OR NOT (bits[17] XOR bits[18]) OR NOT bits[20] THEN error := TRUE; END_IF;
		(* decode minute *)
		minute := 0;
		minute.0 := bits[21];
		minute.1 := bits[22];
		minute.2 := bits[23];
		minute.3 := bits[24];
		IF bits[25] THEN minute := minute + 10; END_IF;
		IF bits[26] THEN minute := minute + 20; END_IF;
		IF bits[27] THEN minute := minute + 40; END_IF;
		IF minute > 59 OR (bits[21] XOR bits[22] XOR bits[23] XOR bits[24] XOR bits[25] XOR bits[26] XOR bits[27] XOR bits[28]) THEN error := TRUE; END_IF;

		(* decode hour *)
		hour := 0;
		hour.0 := bits[29];
		hour.1 := bits[30];
		hour.2 := bits[31];
		hour.3 := bits[32];
		IF bits[33] THEN hour := hour + 10; END_IF;
		IF bits[34] THEN hour := hour +20; END_IF;
		IF hour > 23 OR (bits[29] XOR bits[30] XOR bits[31] XOR bits[32] XOR bits[33] XOR bits[34] XOR bits[35]) THEN error := TRUE; END_IF;

		(* decode day of month *)
		day := 0;
		day.0 := bits[36];
		day.1 := bits[37];
		day.2 := bits[38];
		day.3 := bits[39];
		IF bits[40] THEN day := day + 10; END_IF;
		IF bits[41] THEN day := day + 20; END_IF;
		IF day > 31 THEN error := TRUE; END_IF;

		(* decode day of week *)
		weekday := 0;
		weekday.0 := bits[42];
		weekday.1 := bits[43];
		weekday.2 := bits[44];
		IF weekday > 7 OR weekday < 1 THEN error := TRUE; END_IF;

		(* decode month *)
		month := 0;
		month.0 := bits[45];
		month.1 := bits[46];
		month.2 := bits[47];
		month.3 := bits[48];
		IF bits[49] THEN month := month +10; END_IF;
		IF month > 12 THEN error := TRUE; END_IF;

		(* decode year *)
		year := 0;
		year.0 := bits[50];
		year.1 := bits[51];
		year.2 := bits[52];
		year.3 := bits[53];
		IF bits[54] THEN year := year + 10; END_IF;
		IF bits[55] THEN year := year + 20; END_IF;
		IF bits[56] THEN year := year + 40; END_IF;
		IF bits[57] THEN year := year + 80; END_IF;

		(* check parity for bits 36 to 58 *)
		cnt := 0;
		FOR i := 36 TO 58 DO IF bits[i] THEN cnt := cnt + 1; END_IF; END_FOR;
		IF NOT even(cnt) THEN error := TRUE; END_IF;

		(* time must be valid for two cycles to clear error flag *)
		IF NOT error THEN
			(* set outputs *)
			old_time := mez;
			IF year >= 70 THEN year := year + 1900; ELSE year := year + 2000; END_IF;
			mez := set_DT(year,month,day,hour,minute,0);
			DST := bits[17];
			IF DST THEN
				UTC := DWORD_TO_DT(DT_TO_DWORD(mez) - 7200);
			ELSE
				UTC := DWORD_TO_DT(DT_TO_DWORD(mez) - 3600);
			END_IF

			(* set trigger signal only if the receiver has received 2 successive minutes *)
			IF mez <> old_time + t#1m THEN error := TRUE ; END_IF;
		END_IF;
	END_IF;
END_IF;

(* this portion implements a free running clock which is triggered by the dcf77 signal *)
tz := DWORD_TO_TIME(INT_TO_DWORD(ABS(time_offset))* 3600000);

(* input sdt is copied to utc at first power up *)
IF NOT init THEN
	init := TRUE;
	utc := sdt;
	tp := TRUE;
END_IF;

IF tp THEN
	rtc := utc;
	IF DST AND dst_en THEN
		IF time_offset < 0 THEN	rtc1 := rtc - tz + t#1h; ELSE rtc1 := rtc + tz + t#1h; END_IF;
	ELSE
		IF time_offset < 0 THEN rtc1 := rtc - tz; ELSE rtc1 := rtc + tz; END_IF;
	END_IF;
	sync := TRUE;
	last_sync := last;
	ty := last;
ELSIF rtc > DWORD_TO_DT(0) AND T1 - ty >= t#1s THEN
	rtc := rtc + t#1s;
	rtc1 := rtc1 + t#1s;
	ty := ty + t#1s;
	sync := ty - last_sync < sync_timeout AND last_sync > DWORD_TO_TIME(0);
	weekday := weekday(DT_TO_DATE(rtc1));
	DST := dst_en AND DST(utc);
END_IF;
msec := TIME_TO_INT(t1 - ty);



(* decode information
bits		content
0			Bitwert immer 0
1 bis 14	reserviert für Betriebsinformationen (nicht für DCF77-Nutzer bestimmt)
15			Rufbit für Alarmierung der PTB-Mitarbeiter
			(bis Mai 2003: Bitwert = 0 falls normale Antenne in Verwendung; 1 = Backupantenne)
16			Bitwert = 1 falls ein Wechsel von MEZ nach MESZ oder umgekehrt bevorsteht; Dauer der Anzeige: 1 Stunde
17 + 18	gültige Zeit = MEZ, falls Bit 17=0 und Bit 18=1
			gültige Zeit = MESZ, falls Bit 17=1 und Bit 18=0
19			Bitwert = 1 falls innerhalb den nächsten 59 Minuten eine Schaltsekunde angeordnet ist. Beim Einfügen einer Schaltsekunde wird anstelle der 59. die 60. Sekundenmarke weggelassen und in der 58. erfolgt ausnahmsweise ein Trägerabfall.
20			Startbit für Zeitinformation (immer 1)
21 - 27		1, 2, 4, 8, 10, 20, 40 Minuten (bitweise Addition)
28			Prüfbit (gerade Parität) für die Bits 21-27
29 - 34		1, 2, 4, 8, 10, 20 Stunden (bitweise Addition)
35			Prüfbit (gerade Parität) für die Bits 29-34
36 - 41		Tagesnummer im aktuellen Monat: 1, 2, 4, 8, 10, 20 (bitweise Addition)
42 - 44		Tagesnummer in der aktuellen Woche: 1, 2, 4 (bitweise Addition)
45 - 49		Monatsnummer: 1, 2, 4, 8, 10 (bitweise Addition)
50 - 57		Jahr (zweistellig): 1, 2, 4, 8, 10, 20, 40, 80 (bitweise Addition)
58			Prüfbit (gerade Parität) füR die Bits 36-57

*)
(* revision history

hm 2.feb 2007		rev 1.1
	change wday and dst outputs when there is no dcf reception

hm	26.feb 2007		rev 1.2
	changed statements where t#1h would be substracted from DT.
	under certain conditions the compiler would crash translating this statement

hm	17. sep 2007	rev 1.3
	replaced time() with T_PLC_MS() for compatibility reasons

hm	24. oct 2007	rev 1.4
	changed dst calculation because function dst was upgraded no error in DCF77 only a change in DST

hm	12. nov 2007	rev 1.5
	changed time_offset from time to integer to allow for negative offset time zones

hm	8. dec 2007		rev 1.6
	corrected an error in time_zone calculation

hm 23. jan 2008		rev 1.7
	added sdt input which is used to initialize rtc and rtc1 during first cycle. 
*)
END_FUNCTION_BLOCK

(* POU Time&Date/DST, ST *)
FUNCTION DST : BOOL
VAR_INPUT
	utc : DT;
END_VAR
VAR
	yr : INT;
	yr4 : DWORD;
	ltc: DWORD;
	idate : DWORD;
END_VAR

(*
version 1.2	1 dec 2007
programmer 	hugo
tested by		tobias

this functions returns TRUE IF dst TIME is active 
the FUNCTION calculates automatically for any year betweek 1970 AND 2099 
wheather daylight savings is on OR off 
the summertime calculation is done according to european standards.
dst will become TRUE AT 01:00 utc in the morning FOR the respective days 
AND it will become FALSE after daylight savings TIME is switched back end OF october at 01:00 utc

*)
yr := year(DT_TO_DATE(utc));
ltc := DT_TO_DWORD(utc);
idate := DT_TO_DWORD(set_DT(yr,3,31,1,0,0));
yr4 := SHR(5*yr,2);
IF idate - ((yr4+4) MOD 7)*86400 <= ltc AND idate + (214 - (yr4+1) MOD 7)*86400 > ltc THEN DST := TRUE; ELSE DST := FALSE; END_IF;

(* revision history
hm	4. aug 2006		rev 1.0
	original version

hm	24. okt 2007	rev 1.1
	deleted time_zone_offset input because dst is generally at 01:00 utc and not mesz
	uk starts 01:00 utc and also greece

hm	1. dec 2007		rev 1.2
	changed code to improove performance

*)

(*
Equation used TO calculate the beginning OF European Summer TIME:
Sunday (31 - (5*y/4 + 4) mod 7) March at 01.00 UTC
(valid through 2099, courtesy of Robert H. van Gent, EC).

European Summer Time ends (clocks go back) at 01.00 UTC on

    * 29 October 2006
    * 28 October 2007
    * 26 October 2008

Equation used to calculate the end of European Summer Time:
Sunday (31 - (5*y/4 + 1) mod 7) October at 01.00 UTC
(validity AND credits as above).

*)
END_FUNCTION

(* POU Engineering/control/dead_zone, ST *)
FUNCTION dead_zone : REAL
VAR_INPUT
	X : REAL;
	L : REAL;
END_VAR
VAR
END_VAR

(*
version 1.0	12 Feb 2007
programmer 	hugo
tested by		tobias

dead_zone2 is a linear transfer function which follows a linear function except for x is close to 0.
Y = X if abs(x) > L otherwise its 0.

*)
IF ABS(x) > L THEN
	dead_zone := X;
ELSE
	dead_zone := 0;
END_IF;
END_FUNCTION

(* POU Engineering/control/dead_zone2, ST *)
FUNCTION_BLOCK dead_zone2
VAR_INPUT
	X : REAL;
	L : REAL;
END_VAR
VAR_OUTPUT
	Y: REAL;
END_VAR
VAR
END_VAR

(*
version 1.0	12 Feb 2007
programmer 	hugo
tested by		tobias

dead_zone2 is a linear transfer function which follows a linear function except for x is close to 0.
Y = X if abs(x) > L.
for values of 0 +/. L a hysteresis function will hold the output at + or - L.

*)
IF ABS(x) > L THEN
	Y := X;
ELSIF Y > 0 THEN
	Y := L;
ELSE
	Y := -L;
END_IF;
END_FUNCTION_BLOCK

(* POU Logic/gate logic/DEC_2, ST *)
FUNCTION_BLOCK DEC_2
VAR_INPUT
	D: BOOL;
	A: BOOL;
END_VAR
VAR_OUTPUT
	Q0: BOOL;
	Q1: BOOL;
END_VAR
VAR
END_VAR

(*
version 1.1	3 Mar 2007
programmer 	hugo
tested by		tobias

a bit input will be decoded to the two outputs Q0 or Q1
dependent on the value of A
A=0 decodes to Q0 and A=1 decodes to Q1

*)
Q0 := D AND NOT A;
Q1 := D AND A;

(* revision history
hm 3.3.2007	rev 1.1
	rewritten in ST for better compatibility

*)
END_FUNCTION_BLOCK

(* POU Logic/gate logic/DEC_4, ST *)
FUNCTION_BLOCK DEC_4
VAR_INPUT
	D: BOOL;
	A0: BOOL;
	A1: BOOL;
END_VAR
VAR_OUTPUT
	Q0: BOOL;
	Q1: BOOL;
	Q2: BOOL;
	Q3: BOOL;
END_VAR
VAR
END_VAR

(*
version 1.1	3 Mar 2007
programmer 	hugo
tested by		tobias

a bit input will be decoded to one of the 4 outputs
dependent on the Adress on A0 and A1

executioin TIME on wago 750-841 = 9us
*)
Q0 := D AND NOT A0 AND NOT A1;
Q1 := D AND A0 AND NOT A1;
Q2 := D AND NOT A0 AND A1;
Q3 := D AND A0 AND A1;

(* revision history
hm 3.3.2007	rev 1.1
	rewritten in ST for better compatibility

*)
END_FUNCTION_BLOCK

(* POU Logic/gate logic/DEC_8, ST *)
FUNCTION_BLOCK DEC_8
VAR_INPUT
	D: BOOL;
	A0: BOOL;
	A1: BOOL;
	A2: BOOL;
END_VAR
VAR_OUTPUT
	Q0: BOOL;
	Q1: BOOL;
	Q2: BOOL;
	Q3: BOOL;
	Q4: BOOL;
	Q5: BOOL;
	Q6: BOOL;
	Q7: BOOL;
END_VAR
VAR
END_VAR

(*
version 1.1	3 mar 2007
programmer 	hugo
tested by		tobias

a bit input will be decoded to one of the 8 outputs
dependent on the Adress on A0, A1 and A2

executioin TIME on wago 750-841 = 17us
*)
Q0 := D AND NOT A0 AND NOT A1 AND NOT A2;
Q1 := D AND A0 AND NOT A1 AND NOT A2;
Q2 := D AND NOT A0 AND A1 AND NOT A2;
Q3 := D AND A0 AND A1 AND NOT A2;
Q4 := D AND NOT A0 AND NOT A1 AND A2;
Q5 := D AND A0 AND NOT A1 AND A2;
Q6 := D AND NOT A0 AND A1 AND A2;
Q7 := D AND A0 AND A1 AND A2;

(* revision history
hm 3.3.2007	rev 1.1
	rewritten in ST for better compatibility

*)
END_FUNCTION_BLOCK

(* POU Engineering/signal processing/delay_4, ST *)
FUNCTION_BLOCK delay_4
VAR_INPUT
	in : REAL;
END_VAR
VAR_OUTPUT
	out1 : REAL;
	out2 : REAL;
	out3 : REAL;
	out4 : REAL;
END_VAR
VAR
	temp: REAL;
END_VAR

(*
version 1.1	19 jan 2007
programmer 	hugo
tested by		tobias

this function block delays input values by each programm cycle
after 4 cycles the in value has shifted to the out 4 and will be discarded after the next cycle
the blocks can be cascaded.

*)
out4 := out3;
out3 := out2;
out2 := out1;
out1 := temp;
temp := in;

(* revision history

hm 19.1.2007	rev 1.1
	added variable temp to add 1 delay  for q1

*)
END_FUNCTION_BLOCK

(* POU Building/electrical/dimm_i, ST *)
FUNCTION_BLOCK dimm_i
VAR_INPUT
	set : BOOL;
	in : BOOL;
	rst : BOOL;
END_VAR
VAR_INPUT CONSTANT
	T_debounce : TIME := T#10ms;
	T_reconfig : TIME := T#10s;
	T_on_max : TIME := T#0h;
	T_dimm_start : TIME := T#1s;
	T_dimm: TIME := T#3s;
END_VAR
VAR_OUTPUT
	Q : BOOL := 0;
	out : BYTE := 0;
END_VAR
VAR
	tx : TIME := T#0s;
	last_edge : BOOL;
	state : BYTE := 0;
	edge : BOOL := 0;
	r_edge : BOOL := 0;
	T_on : TIME;
	dimm_up: BOOL;
	last_step : TIME;
	tn: TIME;
END_VAR

(*
version 1.3	15 sep 2007
programmer 	hugo
tested by		tobias

this is an intelligent dimmer interface with an autoset feature for "in" it will automatically detect the type of switch:
low active pulses or high high active pulses are allowd for in.
a configurable debounce timer will debounce input signals
if t_on_max is set to anything other then 0 the output will be turned off after the max on time is reached.
the times for debounce, dimming ramp, wait time before dimming and max on time are all programmable.

the dimmer has outputs Q for on and off and also out with the analog dimm value.

*)
(* read system time *)
tn := DWORD_TO_TIME(T_PLC_MS());;

IF rst THEN
	state := 0;
	Q := FALSE;
	dimm_up := TRUE;
ELSIF set THEN
	state := 0;
	Q := TRUE;
	out := 255;
	dimm_up := FALSE;
	T_on := Tn;
ELSE
	CASE state OF
	(* state 0 wait for activity *)
	0 :	IF (r_edge AND in AND NOT edge) OR (NOT r_edge AND NOT in AND edge) THEN
			IF t_debounce = t#0s THEN state := 2;  ELSE state := 1; END_IF;
			tx := Tn;
			last_edge := in;
		END_IF

	(* state 1 debouncing *)
	1:	IF Tn - T_debounce >= tx THEN
			state := 2;
			tx := Tn;
		END_IF;

	(* state 2 wait for second edge to toggle output *)
	2:	IF Tn - T_dimm_start >= tx THEN
			state := 3;
			tx := Tn;
			(* time to switch elapsed without switching if Q = 0 turn on output and start dimming at 1 *)
			IF NOT Q THEN
				Q := TRUE;
				t_on := tx;
				out := 1;
				dimm_up := TRUE;
			ELSE
				IF out = 255 THEN dimm_up := FALSE; END_IF;
			END_IF;
		ELSIF in XOR edge THEN
			(* wait for edge to toggle output and stop all activity *)
			IF Q THEN
				Q := FALSE;
				state := 0;
			ELSE
				Q := TRUE;
				state := 3;
				IF out = 0 THEN out := 255; END_IF
				IF out = 255 THEN dimm_up := FALSE; END_IF;
				tx := Tn;
				t_on := tx;
			END_IF;
		END_IF;

	(* state 3 entered dimming phase *)
	3:	IF in AND r_edge THEN
			(* generate ramp *)
			tx := Tn;
			IF tx >= last_step + T_dimm / 255 THEN
				last_step := tx;
				IF dimm_up AND out < 255 THEN
					out := out + 1;
					IF out = 255 THEN
						dimm_up := FALSE;
						state := 0;
					END_IF;
				ELSIF NOT dimm_up AND out > 0 THEN
					out := out -1;
					IF out = 0 THEN
						Q := FALSE;
						state := 0;
						dimm_up := TRUE;
					 END_IF;
				 END_IF;
			END_IF;
		ELSE
			dimm_up := NOT dimm_up;
			state := 0;
		END_IF;

	END_CASE;

	(* check for max t_on time and reset output if too long *)
	IF Q AND t_on_max > T#0s AND Tn - t_on_max >= T_on THEN Q := 0; END_IF;

	(* check for reconfig and set R_edge to high for rising edge sensitivity *)
	IF Tn - T_reconfig >= tx THEN R_edge := NOT in; END_IF;

	(* set edge to follow in for next edge detection *)
	edge := in;
END_IF;


(* revision history

hm 22.1.2007		rev 1.1
	deleted unused structure ramp

hm 2.feb 2007		rev 1.2
	changed structure to read time() at the beginning for better time consistency if a higher priorized tak interrupts dimm_i
	added statements in case structure for state 1 to allow for short 1 cycle input pulses

hm 	15.9.2007		rev 1.3
	replaced Time() with T_PLC_MS for compatibility and performance reasons

*)
END_FUNCTION_BLOCK

(* POU Engineering/automation/DRIVER_1, ST *)
FUNCTION_BLOCK DRIVER_1
VAR_INPUT CONSTANT
	Toggle_Mode : BOOL;
	Timeout : TIME;
END_VAR
VAR_INPUT
	SET : BOOL;
	IN : BOOL;
	RST : BOOL;
END_VAR
VAR_OUTPUT
	Q : BOOL;
END_VAR
VAR
	off : TON;
	edge: BOOL;
END_VAR

(*
version 1.0	2 jan 2008
programmer 	hugo
tested by		tobias

driver_1 is a multi purpose driver.
a rising edge on in sets the output high if toggle is flase. while toggle is true, a rising edge on in toggles the output Q.
if a timeout is specified the output q will be reset to false automatically after the timeout has elapsed.
a asynchronous reset and set will force the output high or low respectively.

*)
IF off.Q THEN Q := FALSE; END_IF;
IF rst THEN
	Q := FALSE;
ELSIF set THEN
	Q := TRUE;
ELSIF IN AND NOT edge THEN
	IF toggle_mode THEN q := NOT Q; ELSE q := TRUE; END_IF;
END_IF;
edge := in;
IF timeout > t#0s THEN off(in := Q, PT := Timeout); END_IF;


(* revision history
hm	2. jan 2008		rev 1.0
	original version

*)
END_FUNCTION_BLOCK

(* POU Engineering/automation/DRIVER_4, ST *)
FUNCTION_BLOCK DRIVER_4
VAR_INPUT CONSTANT
	Toggle_Mode : BOOL;
	Timeout : TIME;
END_VAR
VAR_INPUT
	SET : BOOL;
	IN0, IN1, IN2, IN3 : BOOL;
	RST : BOOL;
END_VAR
VAR_OUTPUT
	Q0, Q1, Q2, Q3 : BOOL;
END_VAR
VAR
	d0, d1, d2, d3 : DRIVER_1;
END_VAR

(*
version 1.0	2 jan 2008
programmer 	hugo
tested by		tobias

driver_4 is a 4 channel multi purpose driver.
a rising edge on in? sets the output Q? high if toggle_mode is flase. while toggle_mode is true, a rising edge on in? toggles the output Q?.
if a timeout is specified the output Q? will be reset to false automatically after the timeout has elapsed.
a asynchronous reset and set will force the output high or low respectively.
an asynchronous set will force all outputs high simultaneously

*)
D0(Set:=set, in:=in0, rst:=rst, toggle_mode:=toggle_mode, timeout:=timeout);
D1(Set:=set, in:=in1, rst:=rst, toggle_mode:=toggle_mode, timeout:=timeout);
D2(Set:=set, in:=in2, rst:=rst, toggle_mode:=toggle_mode, timeout:=timeout);
D3(Set:=set, in:=in3, rst:=rst, toggle_mode:=toggle_mode, timeout:=timeout);
Q0 := D0.Q;
Q1 := D1.Q;
Q2 := D2.Q;
Q3 := D3.Q;


(* revision history
hm	2. jan 2008		rev 1.0
	original version

*)
END_FUNCTION_BLOCK

(* POU Logic/gate logic/DWord_of_Byte, ST *)
FUNCTION DWord_of_Byte : DWORD
VAR_INPUT
	B0 : BYTE;
	B1 : BYTE;
	B2 : BYTE;
	B3 : BYTE;
END_VAR
VAR
END_VAR

(*
version 1.1	2 jan 2008
programmer 	hugo
tested by		tobias

this function creates a Dword from 4 individual bytes

*)
DWord_of_Byte := SHL(SHL(SHL(B3,8) OR B2,8) OR B1,8) OR B0;

(* code before rev 1.1
DWord_of_Byte := B3;
DWord_of_Byte := SHL(DWord_of_Byte,8) OR B2;
DWord_of_Byte := SHL(DWord_of_Byte,8) OR B1;
DWord_of_Byte := SHL(DWord_of_Byte,8) OR B0;
*)


(* revision history
hm	24. jan 2007	rev 1.0
	original version

hm 2. jan 2008		rev 1.1
	inproved performance

*)
END_FUNCTION

(* POU String/DWORD_TO_STRF, ST *)
FUNCTION DWORD_TO_STRF : STRING
VAR_INPUT
	IN : DWORD;
	N : INT;
END_VAR
VAR
	L: INT;
	temp: STRING;
END_VAR

(*
version 1.0	26 jan 2007
programmer 	hugo
tested by		tobias

dword_to_strF converts a DWORD, BYTE or Word to a fixed length String.
the string will be filled with leading zeroes to achieve the fixed length, or if too long, the lowest digits will be used.

for example:	dword_to_strf(123,4) = '0123' 
				dword_to_strf(123,2) = '23'
*)
(* convert dword to string first and cut to length N *)
temp := RIGHT(DWORD_TO_STRING(in),N);
L := LEN(temp);
WHILE L < N DO
	temp := CONCAT('0', temp);
	L := L + 1;
END_WHILE;
DWORD_To_STRF := temp;
END_FUNCTION

(* POU XTEST/Baustein Tests/easter_test, ST *)
FUNCTION easter_test : BOOL
VAR_INPUT
END_VAR
VAR
	x: BOOL := TRUE;
END_VAR
x := easter(1980) = d#1980-4-6;
x := easter(1981) = d#1981-4-19 AND x;
x := easter(1982) = d#1982-4-11 AND x;
x := easter(1983) = d#1983-4-3 AND x;
x := easter(1984) = d#1984-4-22 AND x;
x := easter(1985) = d#1985-4-7 AND x;
x := easter(1986) = d#1986-3-30 AND x;
x := easter(1987) = d#1987-4-19 AND x;
x := easter(1988) = d#1988-4-3 AND x;
x := easter(1989) = d#1989-3-26 AND x;
x := easter(1990) = d#1990-4-15 AND x;
x := easter(1991) = d#1991-3-31 AND x;
x := easter(1992) = d#1992-4-19 AND x;
x := easter(1993) = d#1993-4-11 AND x;
x := easter(1994) = d#1994-4-3 AND x;
x := easter(1995) = d#1995-4-16 AND x;
x := easter(1996) = d#1996-4-7 AND x;
x := easter(1997) = d#1997-3-30 AND x;
x := easter(1998) = d#1998-4-12 AND x;
x := easter(1999) = d#1999-4-4 AND x;
x := easter(2000) = d#2000-4-23 AND x;
x := easter(2001) = d#2001-4-15 AND x;
x := easter(2002) = d#2002-3-31 AND x;
x := easter(2003) = d#2003-4-20 AND x;
x := easter(2004) = d#2004-4-11 AND x;
x := easter(2005) = d#2005-3-27 AND x;
x := easter(2006) = d#2006-4-16 AND x;
x := easter(2007) = d#2007-4-8 AND x;
x := easter(2008) = d#2008-3-23 AND x;
x := easter(2009) = d#2009-4-12 AND x;
x := easter(2010) = d#2010-4-4 AND x;
x := easter(2011) = d#2011-4-24 AND x;
x := easter(2012) = d#2012-4-8 AND x;
x := easter(2013) = d#2013-3-31 AND x;
x := easter(2014) = d#2014-4-20 AND x;
x := easter(2015) = d#2015-4-5 AND x;
x := easter(2016) = d#2016-3-27 AND x;
x := easter(2017) = d#2017-4-16 AND x;
x := easter(2018) = d#2018-4-1 AND x;
x := easter(2019) = d#2019-4-21 AND x;
x := easter(2020) = d#2020-4-12 AND x;
x := easter(2021) = d#2021-4-4 AND x;
x := easter(2022) = d#2022-4-17 AND x;
x := easter(2023) = d#2023-4-9 AND x;
x := easter(2024) = d#2024-3-31 AND x;
x := easter(2025) = d#2025-4-20 AND x;
x := easter(2026) = d#2026-4-5 AND x;
x := easter(2027) = d#2027-3-28 AND x;
x := easter(2028) = d#2028-4-16 AND x;
x := easter(2029) = d#2029-4-1 AND x;
x := easter(2030) = d#2030-4-21 AND x;
x := easter(2031) = d#2031-4-13 AND x;
x := easter(2032) = d#2032-3-28 AND x;
x := easter(2033) = d#2033-4-17 AND x;
x := easter(2034) = d#2034-4-9 AND x;
x := easter(2035) = d#2035-3-25 AND x;
x := easter(2036) = d#2036-4-13 AND x;
x := easter(2037) = d#2037-4-5 AND x;
x := easter(2038) = d#2038-4-25 AND x;
x := easter(2039) = d#2039-4-10 AND x;
x := easter(2040) = d#2040-4-1 AND x;
x := easter(2041) = d#2041-4-21 AND x;
x := easter(2042) = d#2042-4-6 AND x;
x := easter(2043) = d#2043-3-29 AND x;
x := easter(2044) = d#2044-4-17 AND x;
x := easter(2045) = d#2045-4-9 AND x;
x := easter(2046) = d#2046-3-25 AND x;
x := easter(2047) = d#2047-4-14 AND x;
x := easter(2048) = d#2048-4-5 AND x;
x := easter(2049) = d#2049-4-18 AND x;
easter_test := X;
END_FUNCTION

(* POU Mathematical/Geometry/ellipse_A, ST *)
FUNCTION ellipse_A : REAL
VAR_INPUT
	R1 : REAL;
	R2 : REAL;
END_VAR
VAR
END_VAR

(*
version 1.0	16 oct 2007
programmer 	hugo
tested by		tobias

ellipse_A calculates the Area of an ellipe based on the two radians R1 and R2


*)
ellipse_A := PI1 * R1 * R2;

(* revision histroy
hm	16. oct 2007	rev 1.0
	original version

*)
END_FUNCTION

(* POU Mathematical/Geometry/ellipse_C, ST *)
FUNCTION ellipse_C : REAL
VAR_INPUT
	R1 : REAL;
	R2 : REAL;
END_VAR
VAR
END_VAR

(*
version 1.0	16 oct 2007
programmer 	hugo
tested by		tobias

ellipse_C calculates the circumference of an ellipe based on the two radians R1 and R2

*)
ellipse_C := PI1 * (3*(R1+R2) - SQRT((3*r1 + R2)*(3*r2 + r1)));

(* revision histroy
hm	16. oct 2007	rev 1.0
	original version

*)
END_FUNCTION

(* POU Engineering/conversion/energy, ST *)
FUNCTION_BLOCK energy
VAR_INPUT
	J : REAL;
	C : REAL;
	Wh : REAL;
END_VAR
VAR_OUTPUT
	YJ : REAL;
	YC : REAL;
	YWh : REAL;
END_VAR
VAR
END_VAR

(*
version 1.0	27 mar 2007
programmer 	hugo
tested by		oscat

this function converts different energy units
any unused input can simply be left open.
different inputs connected at the same time will be added up.
*)
YJ := J + Wh * 3600 + C * 4.1868;
YC := YJ / 4.1868;
YWh := YJ / 3600;

(*
Arbeit, Energie, Joule* J 1 J = 1 N · m = 1 W · s = (1/3,6) E–6 kW · h = 1 kg · m2/s2
Wärmemenge Kilowattstunde kW · h 1 kW · h = 3,6 MJ = 860 kcal
Elektronvolt eV 1 eV = 160,218 92 E–21 J
Erg erg 1 erg = 1E–7 J
Kalorie cal 1 cal = 4,1868 J = 1,163 E–3 W · h
Therm therm 1 therm = 105,50 · 106 J

*)
END_FUNCTION_BLOCK

(* POU String/EXEC, ST *)
FUNCTION EXEC : STRING
VAR_INPUT
	str : STRING;
END_VAR
VAR
	pos: INT;
	R1: REAL;
	R2: REAL;
	operator: STRING;
END_VAR

(*
version 1.2	5. mar. 2008
programmer 	hugo
tested by		tobias

exec executes a mathematical term and returns the result as a string
the term can only be a simple term without brackets and only one operator
allowed operastors are: (+, -, *, /, ^, sqrt, sin, cos, tan).

*)
(* extract both numbers and operator *)
EXEC := UPPERCASE(TRIM(str));

pos := FINDB_NONUM(EXEC);
IF pos > 1 THEN R1 := STRING_TO_REAL(exec); END_IF;
R2 := STRING_TO_REAL(RIGHT(exec,LEN(exec)-pos));
exec := LEFT(exec,pos);
pos := findB_Num(exec);
operator := RIGHT(exec,LEN(exec) - pos);
IF operator = '' AND LEN(str) = 0 THEN
	exec := '';
	RETURN;
ELSIF operator = '' THEN
	exec := str;
	RETURN;
END_IF;
IF operator = '^' THEN
	exec := REAL_TO_STRING(EXPT(R1, R2));
ELSIF operator = 'SQRT' THEN
	exec := REAL_TO_STRING(SQRT(R2));
ELSIF operator = 'SIN' THEN
	EXEC := REAL_TO_STRING(SIN(r2));
ELSIF operator = 'COS' THEN
	exec := REAL_TO_STRING(COS(r2));
ELSIF operator = 'TAN' THEN
	exec := REAL_TO_STRING(TAN(R2));
ELSIF operator = '*' THEN
	exec := REAL_TO_STRING(R1 * R2);
ELSIF operator = '/' THEN
	IF R2 <> 0 THEN exec := REAL_TO_STRING(R1 / R2); ELSE exec := 'ERROR'; END_IF;
ELSIF operator = '+' THEN
	exec := REAL_TO_STRING(r1 + r2);
ELSIF operator = '-' THEN
	exec := REAL_TO_STRING(r1 - r2);
ELSE
	exec := 'ERROR';
END_IF;

(* some systems deliver n. instead of n.0 ! *)
IF RIGHT(EXEC,1) = '.' THEN EXEC := CONCAT(EXEC,'0'); END_IF;



(* revision history

hm 	6.feb 2007		rev 1.1
	cos has to be written in uppercase
	divide by 0 will return an error

hm		5. mar. 2008	rev 1.2
	add a 0 to the string if a '.' is at the end of the string     
*)
END_FUNCTION

(* POU String/UPPERCASE, ST *)
FUNCTION UPPERCASE : STRING
VAR_INPUT
	str : STRING;
END_VAR
VAR
	PT : POINTER TO BYTE;
	pos: INT;
	l: INT;
END_VAR

(*
version 1.1	4. feb 2008
programmer 	hugo
tested by		tobias

uppercase returns str while all letters a..z and ä,ö,ü are converted to uppercase

*)
PT := ADR(UPPERCASE);
uppercase := str;
l := LEN(str);
FOR pos := 1 TO l DO
	pt^ := TO_UPPER(pt^);
	PT := PT + 1;
END_FOR;

(* revision histroy
hm		6.10.2006		rev 1.0
	original release

hm		4. feb. 2008	rev 1.1
	improved performance
	added Ä,Ö,Ü

hm		6. mar 2008	rev 1.2
	added support for exteded Ascii
*)	
END_FUNCTION

(* POU String/TRIM, ST *)
FUNCTION TRIM : STRING
VAR_INPUT
	str : STRING;
END_VAR
VAR
	pos: INT;
END_VAR

(*
version 1.0	6 oct 2006
programmer 	hugo
tested by		tobias

the function deletes all blanks within a string.

*)
TRIM := str;
REPEAT
	pos := FIND(trim,' ');
	trim := REPLACE(trim,'',1,pos);
UNTIL pos = 0	END_REPEAT;


(* revision histroy
hm		6.10.2006		rev 1.0
	original release

*)
END_FUNCTION

(* POU String/FINDB_NONUM, ST *)
FUNCTION FINDB_NONUM : INT
VAR_INPUT
	str : STRING;
END_VAR
VAR
	pos: INT;
	pt : POINTER TO BYTE;
END_VAR

(*
version 1.1	29. feb 2008
programmer 	hugo
tested by		tobias

findB_noNum searches str backwards and returns the last position which is not a number.
a number is characterized by a letter "0..9" or "."

*)
pt := ADR(str) + LEN(str) - 1;
FOR pos := LEN(str) TO 1 BY -1 DO;
	IF NOT((PT^ > 47 AND PT^ < 58) OR PT^ = 46) THEN
		FINDB_NONUM := pos;
		RETURN;
	END_IF;
	PT := PT - 1;
END_FOR;
FINDB_NONUM := 0;


(* revision history
hm		6. oct 2006	rev 1.0
	original version

hm		29. feb 2008	rev 1.1
	improved performance
*)
END_FUNCTION

(* POU String/FINDB_NUM, ST *)
FUNCTION FINDB_NUM : INT
VAR_INPUT
	str : STRING;
END_VAR
VAR
	pos: INT;
	pt : POINTER TO BYTE;
END_VAR

(*
version 1.1	29. feb 2008
programmer 	hugo
tested by		tobias

findB_Num searches str backward and returns the last position of a number
a number is characterized by a letter "0..9" or "."

*)
pt := ADR(str) + LEN(str) - 1;
FOR pos := LEN(str) TO 1 BY -1 DO;
	IF (PT^ > 47 AND PT^ < 58) OR PT^ = 46 THEN
		FINDB_NUM := pos;
		RETURN;
	END_IF;
	PT := PT - 1;
END_FOR;
FINDB_NUM := 0;

(* revision history
hm		6. oct 2006	rev 1.0
	original version

hm		29. feb 2008	rev 1.1
	improved performance
*)
END_FUNCTION

(* POU Building/electrical/F_Lamp, ST *)
FUNCTION_BLOCK F_Lamp
VAR_INPUT
	SWITCH : BOOL;
	DIMM : BYTE := 255;
	Rst : BOOL;
END_VAR
VAR_OUTPUT
	Lamp : BYTE;
	ontime : REAL;
	cycles : REAL;
	Status : BYTE;
END_VAR
VAR_INPUT CONSTANT
	T_no_Dimm : REAL := 100;
	T_Maintenance : REAL := 15000;
END_VAR
VAR
	runtime : ontime;
	maintenance: BOOL;
END_VAR

(*
version 1.1	8 Feb 2007
programmer 	hugo
tested by		tobias

F_Lamp is an interface to flourescent lamps. its main purpose is to protect flourescent lamps from dimming within the first T_NO_DIMM Time.
If Flourescent Lamps are dimmed during the first 100 hours the lifetime of the lamp is reduced dramatically.
The interface also counts ontime and cycles of the lamp for maintanance purposes.

*)
IF rst THEN
	runtime.rst := TRUE;
	runtime();
	runtime.rst := FALSE;
	ontime := runtime.ontime;
	cycles := runtime.cycles;
	maintenance := FALSE;
ELSE
	runtime(in := Switch);
	ontime := runtime.ontime;
	cycles := runtime.cycles;
END_IF;

IF NOT maintenance AND runtime.ontime >= T_maintenance AND T_Maintenance > 0 THEN
	status := 120;
	maintenance := TRUE;
ELSIF Switch THEN
	IF runtime.ontime < T_no_Dimm THEN
		Lamp := 255;
		STATUS := 111;
	ELSE
		Lamp := DIMM;
		status := 112;
	END_IF;
ELSE
	lamp := 0;
	status := 110;
END_IF;
END_FUNCTION_BLOCK

(* POU Mathematical/functions/F_lin, ST *)
FUNCTION F_lin : REAL
VAR_INPUT
	X : REAL;
	A : REAL;
	B : REAL;
END_VAR
VAR
END_VAR

(*
version 1.0	1 sep 2006
programmer 	hugo
tested by		tobias

this function calculates the linear equation f_lin = a*x + b

*)
F_lin := A * X + B;
END_FUNCTION

(* POU Mathematical/functions/F_Lin2, ST *)
FUNCTION F_Lin2 : REAL
VAR_INPUT
	X : REAL;
	X1: REAL;
	Y1 : REAL;
	X2 : REAL;
	Y2 : REAL;
END_VAR
VAR

END_VAR

(*
version 1.0	1 jan 2007
programmer 	hugo
tested by		tobias

this function calculates the linear equation f_lin = a*x + b given by two points x1/y1 and x2/y2.

*)
F_Lin2 := (Y2 - Y1) / (X2 - X1) * X + (Y1 * X1 - Y2 * X1) / (X2 - X1) + Y1;
END_FUNCTION

(* POU Mathematical/functions/F_power, ST *)
FUNCTION F_power : REAL
VAR_INPUT
	a : REAL;
	x : REAL;
	n : REAL;
END_VAR
VAR
END_VAR

(*
version 1.0	1 sep 2006
programmer 	hugo
tested by		tobias

this function calculates the power equation f_power = a*x^n

*)
F_power := a * EXPT(X,N);
END_FUNCTION

(* POU Mathematical/functions/F_quad, ST *)
FUNCTION F_quad : REAL
VAR_INPUT
	X : REAL;
	A : REAL;
	B : REAL;
	C : REAL;
END_VAR
VAR
END_VAR

(*
version 1.0	1 sep 2006
programmer 	hugo
tested by		tobias

this function calculates the quadratic equation f_lin = a*x + b

*)
F_quad := a * X * X + B * X + C;
END_FUNCTION

(* POU XTEST/Ideas/f_sqrt, ST *)
FUNCTION f_sqrt : REAL
VAR_INPUT
	X : REAL;
	A : REAL := 0.005;
END_VAR
VAR
	PTR : POINTER TO DWORD;
	temp: REAL;
END_VAR
(*
IF X > 2 THEN f_sqrt := X/2; ELSE f_sqrt := X; END_IF;
*)
f_sqrt := X;
ptr := ADR(f_sqrt);
ptr^ := 16#5F375A86 - SHR(ptr^,1);

REPEAT
	temp := (f_sqrt + X/f_sqrt)/2;
	f_sqrt := (temp + X/temp)/2;
UNTIL temp - f_sqrt <= A END_REPEAT;





(*

ptr := ADR(X);
ptr^ := 16#5F375A86 - SHR(ptr^,1);

 IF( a > 2.0f )
temp2Wurzel = a/2.0f;
else
temp2Wurzel = a;
do
{
tempWurzel = temp2Wurzel;
temp2Wurzel = (tempWurzel + a/tempWurzel)/2.0f;
}
while( tempWurzel - temp2Wurzel > 0.05f );
RETURN temp2Wurzel;
*)
END_FUNCTION

(* POU Engineering/conversion/F_to_C, ST *)
FUNCTION F_to_C : REAL
VAR_INPUT
	fahrenheit : REAL;
END_VAR
VAR
END_VAR

(*
version 1.1	6. jan 2008
programmer 	hugo
tested BY		tobias

this FUNCTION converts fahrenheit TO celsius

executioin TIME on wago 750-841 = 15us
*)
F_to_C := (fahrenheit -32) * 0.5555555555555;

(* revision history
hm	4. aug 2006		rev 1.0
	original version

hm	6. jan 2008		rev 1.1
	improved performance

*)
END_FUNCTION

(* POU Engineering/conversion/F_to_OM, ST *)
FUNCTION F_to_OM : REAL
VAR_INPUT
	F : REAL;
END_VAR
VAR
END_VAR

(*
version 1.0	22 jan 2007
programmer 	hugo
tested by		tobias

this function converts frequency to Omega F
Omega = 2*PI*F
*)
F_to_OM := PI2 * F;
END_FUNCTION

(* POU Engineering/conversion/F_to_PT, ST *)
FUNCTION F_to_PT : TIME
VAR_INPUT
	F : REAL;
END_VAR
VAR
END_VAR

(*
version 1.0	4 aug 2006
programmer 	hugo
tested by		tobias

this function converts frequency to periode time  
*)
F_to_PT := DWORD_TO_TIME(REAL_TO_DWORD(1/F*1000));
END_FUNCTION

(* POU Engineering/signal processing/FADE, ST *)
FUNCTION_BLOCK FADE
VAR_INPUT
	IN1 : REAL;
	IN2 : REAL;
	F : BOOL;
	TF : TIME;
	rst : BOOL;
END_VAR
VAR_OUTPUT
	Y : REAL;
END_VAR
VAR CONSTANT
	FF : WORD := 65535;
END_VAR
VAR
	rmx : rmp_W;
END_VAR

(*
	version 1.7	26. dec 2007
	programmer 	oscat
	tested BY		oscat

FADE is used to crossfade between the inputs IN1 and IN2. The fade_over time is specified with TF.
When F = TRUE then Y = IN2 after the time TF, and when F = FALSE then Y = IN1.

*)
IF rst THEN
	IF F THEN rmx(set := TRUE, rst := FALSE);	ELSE rmx(rst := TRUE, Set := FALSE); END_IF;
ELSIF F AND (NOT rmx.high) THEN
	rmx(PT := TF, UP := TRUE, en := TRUE, rst := FALSE, set := FALSE);
ELSIF (NOT F) AND (NOT rmx.low) THEN
	rmx(PT := TF, UP := FALSE, en := TRUE, rst := FALSE, set := FALSE);
ELSE
	rmx(En := FALSE, rst := FALSE, set := FALSE);
END_IF;
Y := (WORD_TO_REAL(rmx.out) * in1 + WORD_TO_REAL(FF - rmx.out) * IN2) / FF;

(* revision history
hm	26. dec 2007	rev 1.0
	original version

*)
END_FUNCTION_BLOCK

(* POU XTEST/Performance Test/fb_list, ST *)
FUNCTION_BLOCK fb_list
VAR_INPUT
	num : INT;
	check : BOOL;
END_VAR
VAR
	X1: actuator_2P;
	x2 : actuator_3P;
	x3 : actuator_pump;
	x4 : actuator_UD;
	x5 : click;
	x6 : dimm_i;
	x7 : F_Lamp;
	x8 : Pulse_Length;
	x9 : switch_I;
	x10 : Switch_X;
	x11 : timer_1;
	x12 : timer_2;
	x13 : Boiler;
	x14 : Burner;
	x15 : Heat_temp;
	x16 : legionella;
	x17 : temp_ext;
	x18 : FT_Profile;
	x19 : dead_zone2;
	x20 : FT_deriv;
	x21 : FT_IMP;
	x22 : FT_INT;
	x23 : FT_PID;
	x24 : FT_PT1;
	x25 : FT_PT2;
	x26 : FT_TN16;
	x27 : FT_TN64;
	x28 : FT_TN8;
	x29 : hyst_1;
	x30 : hyst_2;
	x31 : Hyst_3;
	x32 : astro;
	x33 : energy;
	x34 : length;
	x35 : pressure;
	x36 : speed;
	x37 : bar_graph;
	x38 : Calibrate;
	x39 : cycle_time;
	x40 : inc_dec;
	x41 : m_d;
	x42 : m_t;
	x43 : m_tx;
	x44 : ontime;
	x45 : gen_rdm;
	x46 : gen_rmp;
	x47 : gen_sin;
	x48 : gen_sqr;
	x49 : pwm_dc;
	x50 : pwm_pw;
	x51 : rmp_B;
	x52 : rmp_soft;
	x53 : rmp_W;
	x54 : delay;
	x55 : delay_4;
	x56 : SH;
	x57 : SH_1;
	x58 : SH_2;
	x59 : SH_T;
	x60 : stair2;
	x61 : FF_D2E;
	x62 : FF_D4E;
	x63 : FF_DRE;
	x64 : FF_JKE;
	x65 : SHR_4E;
	x66 : SHR_4UDE;
	x67 : SHR_8PLE;
	x68 : SHR_8UDE;
	x69 : LTCH;
	x70 : LTCH_4;
	x71 : Byte_to_Bit;
	x72 : DEC_2;
	x73 : DEC_4;
	x74 : DEC_8;
	x75 : B_TRIG;
	x76 : B_TRIG;
	x77 : CLK_N;
	x78 : CLK_N;
	x79 : CLK_N;
	x80 : clk_div;
	x81 : CLK_Prg;
	x82 : CLK_Pulse;
	x83 : D_Trig;
	x84 : gen_bit;
	x85 : gen_SQ;
	x86 : sequence_4;
	x87 : sequence_8;
	x88 : TP_R;
	x89 : FIFO_16;
	x90 : FIFO_32;
	x91 : STACK_16;
	x92 : STACK_32;
	x93 : matrix;
	x94 : FT_avg;
	x95 : FT_min_max;
	x96 : FT_rmp;
	x97 : ESR_collect;
	x98 : ESR_MON_B8;
	x99 : ESR_MON_R4;
	x100 : ESR_MON_X8;
	x101 : DCF77;
	x102 : holiday;
	x103: Ltime;
	x104 : sun_pos;
	x105 : sun_time;
END_VAR
IF num < 10 THEN
	CASE num OF
	1 : IF check THEN RETURN; ELSE X1; END_IF;
	2 : IF check THEN RETURN; ELSE X2; END_IF;
	3 : IF check THEN RETURN; ELSE X3; END_IF;
	4 : IF check THEN RETURN; ELSE X4; END_IF;
	5 : IF check THEN RETURN; ELSE X5; END_IF;
	6 : IF check THEN RETURN; ELSE X6; END_IF;
	7 : IF check THEN RETURN; ELSE X7; END_IF;
	8 : IF check THEN RETURN; ELSE X8; END_IF;
	9 : IF check THEN RETURN; ELSE X9; END_IF;
	END_CASE;
ELSIF num < 20 THEN
	CASE num OF
	10 : IF check THEN RETURN; ELSE X10; END_IF;
	11 : IF check THEN RETURN; ELSE X11; END_IF;
	12 : IF check THEN RETURN; ELSE X12; END_IF;
	13 : IF check THEN RETURN; ELSE X13; END_IF;
	14 : IF check THEN RETURN; ELSE X14; END_IF;
	15 : IF check THEN RETURN; ELSE X15; END_IF;
	16 : IF check THEN RETURN; ELSE X16; END_IF;
	17 : IF check THEN RETURN; ELSE X17; END_IF;
	18 : IF check THEN RETURN; ELSE X18; END_IF;
	19 : IF check THEN RETURN; ELSE X19; END_IF;
	END_CASE;
ELSIF num < 30 THEN
	CASE num OF
	20 : IF check THEN RETURN; ELSE X20; END_IF;
	21 : IF check THEN RETURN; ELSE X21; END_IF;
	22 : IF check THEN RETURN; ELSE X22; END_IF;
	23 : IF check THEN RETURN; ELSE X23; END_IF;
	24 : IF check THEN RETURN; ELSE X24; END_IF;
	25 : IF check THEN RETURN; ELSE X25; END_IF;
	26 : IF check THEN RETURN; ELSE X26; END_IF;
	27 : IF check THEN RETURN; ELSE X27; END_IF;
	28 : IF check THEN RETURN; ELSE X28; END_IF;
	29 : IF check THEN RETURN; ELSE X29; END_IF;
	END_CASE;
ELSIF num < 40 THEN
	CASE num OF
	30 : IF check THEN RETURN; ELSE X30; END_IF;
	31 : IF check THEN RETURN; ELSE X31; END_IF;
	32 : IF check THEN RETURN; ELSE X32; END_IF;
	33 : IF check THEN RETURN; ELSE X33; END_IF;
	34 : IF check THEN RETURN; ELSE X34; END_IF;
	35 : IF check THEN RETURN; ELSE X35; END_IF;
	36 : IF check THEN RETURN; ELSE X36; END_IF;
	37 : IF check THEN RETURN; ELSE X37; END_IF;
	38 : IF check THEN RETURN; ELSE X38; END_IF;
	39 : IF check THEN RETURN; ELSE X39; END_IF;
	END_CASE;
ELSIF num < 50 THEN
	CASE num OF
	40 : IF check THEN RETURN; ELSE X40; END_IF;
	41 : IF check THEN RETURN; ELSE X41; END_IF;
	42 : IF check THEN RETURN; ELSE X42; END_IF;
	43 : IF check THEN RETURN; ELSE X43; END_IF;
	44 : IF check THEN RETURN; ELSE X44(IN := TRUE); END_IF;
	45 : IF check THEN RETURN; ELSE X45; END_IF;
	46 : IF check THEN RETURN; ELSE X46; END_IF;
	47 : IF check THEN RETURN; ELSE X47; END_IF;
	48 : IF check THEN RETURN; ELSE X48; END_IF;
	49 : IF check THEN RETURN; ELSE X49; END_IF;
	END_CASE;
ELSIF num < 60 THEN
	CASE num OF
	50 : IF check THEN RETURN; ELSE X50; END_IF;
	51 : IF check THEN RETURN; ELSE X51; END_IF;
	52 : IF check THEN RETURN; ELSE X52; END_IF;
	53 : IF check THEN RETURN; ELSE X53; END_IF;
	54 : IF check THEN RETURN; ELSE X54; END_IF;
	55 : IF check THEN RETURN; ELSE X55; END_IF;
	56 : IF check THEN RETURN; ELSE X56; END_IF;
	57 : IF check THEN RETURN; ELSE X57; END_IF;
	58 : IF check THEN RETURN; ELSE X58; END_IF;
	59 : IF check THEN RETURN; ELSE X59; END_IF;
	END_CASE;
ELSIF num < 70 THEN
	CASE num OF
	60 : IF check THEN RETURN; ELSE X60; END_IF;
	61 : IF check THEN RETURN; ELSE X61; END_IF;
	62 : IF check THEN RETURN; ELSE X62; END_IF;
	63 : IF check THEN RETURN; ELSE X63; END_IF;
	64 : IF check THEN RETURN; ELSE X64; END_IF;
	65 : IF check THEN RETURN; ELSE X65; END_IF;
	66 : IF check THEN RETURN; ELSE X66; END_IF;
	67 : IF check THEN RETURN; ELSE X67; END_IF;
	68 : IF check THEN RETURN; ELSE X68; END_IF;
	69 : IF check THEN RETURN; ELSE X69; END_IF;
	END_CASE;
ELSIF num < 80 THEN
	CASE num OF
	70 : IF check THEN RETURN; ELSE X70; END_IF;
	71 : IF check THEN RETURN; ELSE X71; END_IF;
	72 : IF check THEN RETURN; ELSE X72; END_IF;
	73 : IF check THEN RETURN; ELSE X73; END_IF;
	74 : IF check THEN RETURN; ELSE X74; END_IF;
	75 : IF check THEN RETURN; ELSE X75; END_IF;
	76 : IF check THEN RETURN; ELSE X76; END_IF;
	77 : IF check THEN RETURN; ELSE X77; END_IF;
	78 : IF check THEN RETURN; ELSE X78; END_IF;
	79 : IF check THEN RETURN; ELSE X79; END_IF;
	END_CASE;
ELSIF num < 90 THEN
	CASE num OF
	80 : IF check THEN RETURN; ELSE X80; END_IF;
	81 : IF check THEN RETURN; ELSE X81; END_IF;
	82 : IF check THEN RETURN; ELSE X82; END_IF;
	83 : IF check THEN RETURN; ELSE X83; END_IF;
	84 : IF check THEN RETURN; ELSE X84; END_IF;
	85 : IF check THEN RETURN; ELSE X85; END_IF;
	86 : IF check THEN RETURN; ELSE X86; END_IF;
	87 : IF check THEN RETURN; ELSE X87; END_IF;
	88 : IF check THEN RETURN; ELSE X88; END_IF;
	89 : IF check THEN RETURN; ELSE X89; END_IF;
	END_CASE;
ELSIF num < 100 THEN
	CASE num OF
	90 : IF check THEN RETURN; ELSE X90; END_IF;
	91 : IF check THEN RETURN; ELSE X91; END_IF;
	92 : IF check THEN RETURN; ELSE X92; END_IF;
	93 : IF check THEN RETURN; ELSE X93; END_IF;
	94 : IF check THEN RETURN; ELSE X94; END_IF;
	95 : IF check THEN RETURN; ELSE X95; END_IF;
	96 : IF check THEN RETURN; ELSE X96; END_IF;
	97 : IF check THEN RETURN; ELSE X97; END_IF;
	98 : IF check THEN RETURN; ELSE X98; END_IF;
	99 : IF check THEN RETURN; ELSE X99; END_IF;
	END_CASE;
ELSIF num < 110 THEN
	CASE num OF
	100 : IF check THEN RETURN; ELSE X100; END_IF;
	101 : IF check THEN RETURN; ELSE X101; END_IF;
	102 : IF check THEN RETURN; ELSE X102; END_IF;
	103 : IF check THEN RETURN; ELSE X103; END_IF;
	104 : IF check THEN RETURN; ELSE X104; END_IF;
	105 : IF check THEN RETURN; ELSE X105; END_IF;
	END_CASE;
END_IF;
END_FUNCTION_BLOCK

(* POU Building/electrical/switch_I, ST *)
FUNCTION_BLOCK switch_I
VAR_INPUT
	set : BOOL;
	in : BOOL;
	rst : BOOL;
END_VAR
VAR_INPUT CONSTANT
	T_debounce : TIME := T#10ms;
	T_reconfig : TIME := T#1s;
	T_on_max : TIME := T#0h;
END_VAR
VAR_OUTPUT
	Q : BOOL := 0;
END_VAR
VAR
	state : BYTE := 0;
	edge : BOOL := 0;
	r_edge : BOOL := 0;
	T_on : TIME;
	tx: TIME;
END_VAR

(*
version 1.1	15 sep 2007
programmer 	oscat
tested by		tobias

this is an intelligent switch interface which has an autodetect feature for in and it will detect the type of switch connected automatically
the input can be connected to low active pulses, high active pulses and on/off switch.
it will automatically adjust to the correct type without manual adjustment
a configurable debounce timer will debounce input signals
if t_on_max is set to anything other then 0 the output will be turned off after the max on time is reached.

*)
(* read system time *)
tx := DWORD_TO_TIME(T_PLC_MS());

(* asynchronous set and reset first *)
IF set AND NOT rst THEN
	Q := 1;
	T_on := tx;
ELSIF rst THEN
	Q := 0;
(* check FOR input edge AND start debounce timer *)
ELSIF (in XOR edge) AND NOT (state = 1) THEN
	state := 1;
	T_on := Tx;
(* edge was detected and debounce time elapsed *)
ELSIF (state = 1) AND (Tx - t_debounce >= T_on) THEN
	state := 2;
	(* react on rising or falling edge depending on r_edge *)
	IF r_edge XOR in THEN Q := NOT Q; END_IF;
(* wait for T_reconfig and adjust r_edge *)
ELSIF state = 2 AND Tx - t_reconfig >= T_on THEN
	r_edge := in;
END_IF;
IF Q AND T_on_max > t#0ms AND Tx >= T_on + T_on_max THEN
	Q := FALSE;
END_IF;
edge := in;

(* revision history

hm	4 aug 2006	rev 1.0
	original version

hm	15.9.2007	rev 1.1
	replaced Time() with T_PLC_MS for compatibility and performance reasons

*)
END_FUNCTION_BLOCK

(* POU Building/electrical/Switch_X, ST *)
FUNCTION_BLOCK Switch_X
VAR_INPUT
	IN1 : BOOL;
	IN2 : BOOL;
	IN3 : BOOL;
	IN4 : BOOL;
	IN5 : BOOL;
	IN6 : BOOL;
END_VAR
VAR_OUTPUT
	Q1 : BOOL;
	Q2 : BOOL;
	Q3 : BOOL;
	Q4 : BOOL;
	Q5 : BOOL;
	Q6 : BOOL;
	Q31 : BOOL;
	Q41 : BOOL;
	Q51 : BOOL;
	Q61 : BOOL;
	Q32 : BOOL;
	Q42 : BOOL;
	Q52 : BOOL;
	Q62 : BOOL;
END_VAR
VAR_INPUT CONSTANT
	t_debounce : TIME := t#50ms;
END_VAR
VAR
	init : BOOL;
	T1, T2, T3, T4, T5, T6 : TOF;
	tx: TIME;
	x1: BOOL;
	x2: BOOL;
	E1, E2 : BOOL;
END_VAR

(*
version 1.0	15 Feb 2007
programmer 	oscat
tested by		tobias

*)
(* initialize on startup *)
IF NOT init THEN
	init := TRUE;
	IF t_debounce < t#50ms THEN tx := t#50ms; ELSE tx := t_debounce; END_IF;
	T1(PT := Tx);
	T2(PT := Tx);
	T3(PT := Tx);
	T4(PT := Tx);
	T5(PT := Tx);
	T6(PT := Tx);
ELSE
	Q1 := FALSE;
	Q2 := FALSE;
	Q3 := FALSE;
	Q4 := FALSE;
	Q5 := FALSE;
	Q6 := FALSE;
	Q31 := FALSE;
	Q41 := FALSE;
	Q51 := FALSE;
	Q61 := FALSE;
	Q32 := FALSE;
	Q42 := FALSE;
	Q52 := FALSE;
	Q62 := FALSE;
END_IF;

(* read inputs and debounce *)
	T1(IN := IN1);
	T2(IN := IN2);
	T3(IN := IN3);
	T4(IN := IN4);
	T5(IN := IN5);
	T6(IN := IN6);

(* detect edge of IN1 and IN2 *)
IF t1.Q AND NOT E1 THEN X1 := TRUE; END_IF;
IF t2.Q AND NOT E2 THEN X2 := TRUE; END_IF;

IF t1.Q THEN
	IF t3.q THEN
		q31 := TRUE;
		X1 := FALSE;
	ELSIF t4.q THEN
		q41 := TRUE;
		X1 := FALSE;
	ELSIF t5.q THEN
		q51 := TRUE;
		X1 := FALSE;
	ELSIF t6.q THEN
		q61 := TRUE;
		X1 := FALSE;
	END_IF;
ELSIF t2.Q THEN
	IF t3.q THEN
		q32 := TRUE;
		X2 := FALSE;
	ELSIF t4.q THEN
		q42 := TRUE;
		X2 := FALSE;
	ELSIF t5.q THEN
		q52 := TRUE;
		X2 := FALSE;
	ELSIF t6.q THEN
		q62 := TRUE;
		X2 := FALSE;
	END_IF;
(* in1 was active alone *)
ELSIF NOT T1.Q AND E1 AND X1 THEN
	Q1 := TRUE;
	X1 := FALSE;
ELSIF NOT T2.Q AND E2 AND X2 THEN
	Q2 := TRUE;
	X2 := FALSE;
ELSIF T3.Q THEN
	Q3 := TRUE;
ELSIF T4.Q THEN
	Q4 := TRUE;
ELSIF T5.Q THEN
	Q5 := TRUE;
ELSIF T6.Q THEN
	Q6 := TRUE;
END_IF;

(* save state of in1 and in2 *)
E1 := T1.Q;
E2 := T2.Q;
END_FUNCTION_BLOCK

(* POU Building/electrical/timer_1, ST *)
FUNCTION_BLOCK timer_1
VAR_INPUT
	DT_in : DT;
	start_time : TOD;
	duration : TIME;
	start_day : INT := 0;
END_VAR
VAR_OUTPUT
	Q : BOOL;
END_VAR
VAR
	dat : DATE;
	day : INT;
	tmp : DT;
	stop : DT;
	last_dat: DATE;
END_VAR

(*
version 1.6	17. jan 2008
programmer 	oscat
tested by		tobias

this is a simple timer that generates an output pulse once a day if start_day = 0.
if start_day is a number from 1 .. 7 then a output pulse is generated for the respective weekday 1 = monday.
the output pulse width can be programmed, if set to 0 a pulse is generated for one cycle only.

*)
(* calculate the current weekday and date *)
dat := DT_TO_DATE(dt_in);
tmp := DATE_TO_DT(dat) + duration + TOD_TO_TIME(start_time);
IF start_day = 0 THEN day := 0; ELSE day := weekday(dat); END_IF;

(* check if current day is active and start condition is met *)
IF NOT Q AND day = start_day AND DT_TO_TOD(dt_in) >= start_time AND last_dat < dat AND dt_in <= tmp THEN
	Q := TRUE;
	last_dat := dat;
	stop := tmp;
ELSIF dt_in >= stop THEN
	Q := FALSE;
END_IF;

(* code before rev 1.6
tx := DWORD_TO_TIME(T_PLC_MS());

IF NOT init THEN
	init := TRUE;
	last_check := tx - t#100ms;
END_IF;

IF tx - last_check >= T#100ms THEN
	dat := DT_TO_DATE(dt_in);
	IF NOT Q AND (start_day = 0 OR start_day = weekday(dat)) AND dat <> last AND DT_TO_TOD(dt_in) >= start_time THEN
		Q := TRUE;
		last := dat;
		pulse_start := tx;
	ELSIF Q AND tx - pulse_start >= duration THEN
		Q := FALSE;
	END_IF;
	last_check := tx;
END_IF;
*)

(*
1.12.2006 hm		rev 1.1
	corrected an error with pulse width = 0.

25.12.2006 hm	rev 1.2
	corrected an error when timer overflows.

14.apr 2007 hm	rev 1.3
	corrected an error while while output would not go active when start year would be 1970.
	increase accuracy by checking every 100ms
	added init section to compensate for timer overflow

15.9.2007	hm		rev 1.4
	replaced Time() with T_PLC_MS for compatibility and performance reasons

hm	1. okt 2007		rev 1.5
	corrected an error while output would not stay active over midnight.

hm	17. jan 2008	rev 1.6
	New code with better performance  
	Output is now only active during the time of day it is supposed to 
	no pulse is generated at power up

*)
END_FUNCTION_BLOCK

(* POU Building/HLK/Heat_temp, ST *)
FUNCTION_BLOCK Heat_temp
VAR_INPUT
	T_ext : REAL;
	Offset : REAL;
	t_req : REAL;
END_VAR
VAR_INPUT CONSTANT
	TY_max : REAL := 70;
	TY_min : REAL := 20;
	T_int : REAL := 20;
	TY_config : REAL := 50;
	T_ext_config : REAL := -15;
	C : REAL := 1.33;
END_VAR
VAR_OUTPUT
	Ty : REAL;
END_VAR
VAR
END_VAR

(*
version 1.0	27 jan 2007
programmer 	hugo
tested by		tobias

Heat_Temp calculates a heat characteristic based on the formula: tv=ti+(tvmax-ti)*((ti-tau)/(ti-taumin))^(1/n)
while
tv necessary heating temperature.
ti internal room temperature (20°C)
tau current external temperature
external temperature to determine characteristics
C exponent for heating system (normally 1,33 or 1,1 for floor heating)

The two additional inputs TY_min and TY_max set limits for the output TY, while an offset inputs allows to rise or lower the room temperature.

*)
IF t_ext > t_int + Offset THEN
	ty := t_int + offset;
ELSE
Ty := T_int - offset + (TY_config - T_int) * EXPT((T_int - offset - T_ext) / (T_int - offset - T_ext_config),1 / C);
END_IF;
IF t_req > ty THEN ty := t_req; END_IF;
ty := LIMIT(TY_min, ty, TY_max);



(*

tv=ti+(tvmax-ti)*((ti-tau)/(ti-taumin))^(1/n)

tv aktuelle Vorlauftemp.
ti Raumtemperatur innen (20°C)
tau aktuelle Außentemperatur
taumin minimale Außentemperatur -12°C oder -15°C
n Heizkörperexponent (meistens 1,33)
Fußbodenheizung = 1,1
Wandheizung 1,3

Normen z. B. DIN 4703, DIN 4725 oder die Literatur, z. B Recknagel Abschnitt 1.3.5.

*)
END_FUNCTION_BLOCK

(* POU Building/HLK/legionella, ST *)
FUNCTION_BLOCK legionella
VAR_INPUT
	manual : BOOL;
	temp_boiler : REAL;
	temp_return : REAL := 100;
	DT_in: DT;
	rst : BOOL;
END_VAR
VAR_INPUT CONSTANT
	T_start: TOD := tod#03:00:00;
	day : INT := 7;
	temp_set : REAL := 70;
	temp_offset : REAL := 10;
	temp_hys : REAL := 5;
	t_max_heat: TIME := t#10m;
	t_max_ret : TIME := t#10m;
	tp_0: TIME := t#5m;
	tp_1: TIME := t#5m;
	tp_2: TIME := t#5m;
	tp_3: TIME := t#5m;
	tp_4: TIME := t#5m;
	tp_5: TIME := t#5m;
	tp_6: TIME := t#5m;
	tp_7: TIME := t#5m;
END_VAR
VAR_OUTPUT
	Heat : BOOL;
	pump : BOOL;
	valve0 : BOOL;
	valve1 : BOOL;
	valve2 : BOOL;
	valve3 : BOOL;
	valve4 : BOOL;
	valve5 : BOOL;
	valve6 : BOOL;
	valve7 : BOOL;
	run: BOOL;
	Status : BYTE;
END_VAR
VAR
	X1: timer_1;
	x2: sequence_8;
	x3: hyst_1;
	init: BOOL;
END_VAR

(*
version 1.1	17. jan 2007
programmer 	oscat
tested by		hans

Legionella is a complete sequencer for up to 8 hot water lines that need to be sterilzed periodically.
legionella needs a DT input with the appropriate time, usually gererated by the rtc of the system. for system independence this time is connected externally.
T_start is the time when sterilazation should be started and day is the day_of_week when it should be performed (1=Monday and 7=sunday).
so sterilazation is autioimatically performed once a week at a specified time.
temp_set and temp_hys and temp_offset specify the boiler temperatur nedded for sterilization. as a defaut Temp_set is set to 70 deg C and Temp_hys is set to 5 deg C and temp_offset is 10 deg C.
a temp boiler input reads the boiler temperature of the hot water tank.
after a start pulse is gererated by the weekly timer or a manual test input the sequence is started:
1. the boiler is heated to temp_set + temp_offset + temp_hys = 85 deg C unless chaged at setup.
	the heat output is turned on and tells the heater to turn heating on. if the temp is not reached for a time of t_max_heat (10 min) the error output is set and the sequence is stopped.
2. after the specified temperature is reached, the output valve0 and pump is turned on and starts sterilization of line0 until temp_return has reached temp_set and continues to sterilize for a time of tp_0 (5 min default).
	if tmep_set is not reached at the temp_return_input then the error output is set and the sequence will be stopped.
	if there is no temp sensor for temp_return (the temperature at the return point for the circulation pump pls set this imput to a value greater then temp_set (by default use 100 deg C).
	in this case sterilization is performed for the default times without monitoring the return temp.
3. this sequence is repeated for up to valves.

connection scheme:

temp_boiler:	input oif the boiler temperature sensor.
temp_hys:		config value for the heater hysteresis, preset to 5 deg C.
temp_offset:	config value for the heater temp_offset against temp_set, preset to 10 deg C.
temp_set:		config value for the specified sterilization temperature, preset to 70 deg C.
temp_return:	input of the circulation return line temperature sensor, if not availabe set this value to 100 deg C.
manual:		manual input to start the sterilization by hand for diagnostic purposes, rising edge active, leave low for automatic operation.
DT_in:			date,time input supplied by a external real time clock.
T_start:		time of day when the sterilization should be started.
day:			config value for day of week when the process should be started, preset to sunday.
t_max_hest:	tmax time to be needed for the heater to heat the hot water tank to the specified value, preset to 10 min.

*)
(* startup initialization *)
IF NOT init THEN
	init := TRUE;
	X1.start_day := day;
	X1.start_time := T_start;
	X3.low := Temp_offset + temp_set;
	X3.high := Temp_hys + X3.low;
	X2.wait0 := T_max_heat;
	X2.delay0 := TP_0;
	X2.delay1 := TP_1;
	X2.delay2 := TP_2;
	X2.delay3 := TP_3;
	X2.delay4 := TP_4;
	X2.delay5 := TP_5;
	X2.delay6 := TP_6;
	X2.delay7 := TP_7;
	X2.wait1 := T_max_ret;
	X2.wait2 := T_max_ret;
	X2.wait3 := T_max_ret;
	X2.wait4 := T_max_ret;
	X2.wait5 := T_max_ret;
	X2.wait6 := T_max_ret;
	X2.wait7 := T_max_ret;
	X2();
END_IF;

(* oerational code *)
X1(DT_in := DT_in);
IF X1.Q OR manual OR x2.run THEN
	X3(in := temp_boiler);
	X2.in0 := X3.Q OR x3.win;
	X2.in1 := temp_return >= temp_set;
	X2.in2 := x2.in1;
	X2.in3 := x2.in1;
	X2.in4 := x2.in1;
	X2.in5 := x2.in1;
	X2.in6 := x2.in1;
	X2.in7 := x2.in1;
	X2.rst := rst;
	X2(start := X1.Q OR manual);
	run := x2.run;
	pump := x2.any;
	Heat := NOT X3.Q AND x2.run;
	valve0 := X2.Q0;
	valve1 := X2.Q1;
	valve2 := X2.Q2;
	valve3 := X2.Q3;
	valve4 := X2.Q4;
	valve5 := X2.Q5;
	valve6 := X2.Q6;
	valve7 := X2.Q7;
	pump := X2.any;
	status := X2.status;
ELSE;
	X2(start :=0);
	status := x2.status;
END_IF;

(* revision history

hm 17.jan 2007	rev 1.1
	rewritten to st for higher performance
	changes eeror output to esr compatible status output
*)
END_FUNCTION_BLOCK

(* POU Logic/generators/sequence_8, ST *)
FUNCTION_BLOCK sequence_8
VAR_INPUT
	in0 : BOOL := TRUE;
	in1 : BOOL := TRUE;
	in2 : BOOL := TRUE;
	in3 : BOOL := TRUE;
	in4 : BOOL := TRUE;
	in5 : BOOL := TRUE;
	in6 : BOOL := TRUE;
	in7 : BOOL := TRUE;
	start : BOOL;
	rst : BOOL;
	wait0 : TIME := t#0s;
	delay0 : TIME := t#0s;
	wait1 : TIME := t#0s;
	delay1 : TIME := t#0s;
	wait2 : TIME := t#0s;
	delay2 : TIME := t#0s;
	wait3 : TIME := t#0s;
	delay3 : TIME := t#0s;
	wait4 : TIME := t#0s;
	delay4 : TIME := t#0s;
	wait5 : TIME := t#0s;
	delay5 : TIME := t#0s;
	wait6 : TIME := t#0s;
	delay6 : TIME := t#0s;
	wait7 : TIME := t#0s;
	delay7 : TIME := t#0s;
END_VAR
VAR_INPUT CONSTANT
	stop_on_error : BOOL := FALSE;
END_VAR
VAR_OUTPUT
	Q0 : BOOL;
	Q1 : BOOL;
	Q2 : BOOL;
	Q3 : BOOL;
	Q4 : BOOL;
	Q5 : BOOL;
	Q6 : BOOL;
	Q7 : BOOL;
	any : BOOL;
	run: BOOL;
	step : INT := -1;
	status : BYTE;
END_VAR
VAR
	last : TIME;
	edge : BOOL;
	tx: TIME;
	init: BOOL;
END_VAR

(*
version 1.4	17 sep 2007
programmer 	oscat
tested by		hans

sequence_8 enables run when a low to high transition is present on start.
a low to high transition on start will restart the sequencer at any time while a rst will hold the sequencer in reset while true.
after run is enabled with a rising edge on start the sequencer waits for wait0 on in0 to enable q0 which stays on for delay0.
the next cycle starts with wait1, continues with delay 1 and so on...
if an edge is not detected during the wait period, the sequencer will then display the error number on the status output.
The status numbers are 1 .. 8 for erros in step 0..7.
after the last step that sets q7, the sequencer leaves q7 on for delay7 and then resets to the initial state.
a step output will indicate the current step of the sequencer and will also be present with a fault condition.
after the first output is turened on the sequencer switches from q0 to q1 and so on, at any time there is only one output enabled.
if an input signal is not detected during a wait period, the sequencer will display the error number ( 1 for in0, 2 for in1 .... ).
when an error is present and the config variable stop_on_error is set then the sequencer will stop. otherwise it will continue.
The status output will also display 110 for waiting and 111 sequece running.

*)
(* read sps timer *)
tx := DWORD_TO_TIME(T_PLC_MS());

(* initialize on startup *)
IF NOT init THEN
	last := tx;
	init := TRUE;
	status := 110;
END_IF;

(* asynchronous reset *)
IF rst THEN
	step := -1;
	Q0 := 0;
	Q1 := 0;
	Q2 := 0;
	Q3 := 0;
	Q4 := 0;
	Q5 := 0;
	Q6 := 0;
	Q7 := 0;
	status := 110;
	run := 0;

(* edge on start input restarts the sequencer *)
ELSIF start AND NOT edge THEN
	step := 0;
	last := tx;
	status := 111;
	Q0 := 0;
	Q1 := 0;
	Q2 := 0;
	Q3 := 0;
	Q4 := 0;
	Q5 := 0;
	Q6 := 0;
	Q7 := 0;
	run := 1;
END_IF;
edge := start;

(* check if stop on error is necessary *)
IF status > 0 AND status < 100 AND stop_on_error THEN RETURN; END_IF;

(* sequence is running *)
IF run AND step = 0 THEN
	IF NOT q0 AND in0 AND tx - last <= wait0 THEN
		Q0 := TRUE;
		last := tx;
	ELSIF NOT q0 AND tx - last > wait0 THEN
		status := 1;
		run := FALSE;
	ELSIF q0 AND tx - last >= delay0 THEN
		step := 1;
		last := tx;
	END_IF;
END_IF;
IF run AND step = 1 THEN
	IF NOT q1 AND in1 AND tx - last <= wait1 THEN
		Q0 := FALSE;
		Q1 := TRUE;
		last := tx;
	ELSIF NOT q1 AND Tx - last > wait1 THEN
		status := 2;
		q0 := FALSE;
		run := FALSE;
	ELSIF q1 AND tx - last >= delay1 THEN
		step := 2;
		last := tx;
	END_IF;
END_IF;
IF run AND step = 2 THEN
	IF NOT q2 AND in2 AND tx - last <= wait2 THEN
		Q1 := FALSE;
		Q2 := TRUE;
		last := tx;
	ELSIF NOT q2 AND Tx - last > wait2 THEN
		status := 3;
		q1 := FALSE;
		run := FALSE;
	ELSIF q2 AND tx - last >= delay2 THEN
		step := 3;
		last := tx;
	END_IF;
END_IF;
IF run AND step = 3 THEN
	IF NOT q3 AND in3 AND tx - last <= wait3 THEN
		Q2 := FALSE;
		Q3 := TRUE;
		last := tx;
	ELSIF NOT q3 AND Tx - last > wait3 THEN
		status := 4;
		q2 := FALSE;
		run := FALSE;
	ELSIF q3 AND tx - last >= delay3 THEN
		step := 4;
		last := tx;
	END_IF;
END_IF;
IF run AND step = 4 THEN
	IF NOT q4 AND in4 AND tx - last <= wait4 THEN
		Q3 := FALSE;
		Q4 := TRUE;
		last := tx;
	ELSIF NOT q4 AND Tx - last > wait4 THEN
		status := 5;
		q3 := FALSE;
		run := FALSE;
	ELSIF q4 AND tx - last >= delay4 THEN
		step := 5;
		last := tx;
	END_IF;
END_IF;
IF run AND step = 5 THEN
	IF NOT q5 AND in5 AND tx - last <= wait5 THEN
		Q4 := FALSE;
		Q5 := TRUE;
		last := tx;
	ELSIF NOT q5 AND Tx - last > wait5 THEN
		status := 6;
		q4 := FALSE;
		run := FALSE;
	ELSIF q5 AND tx - last >= delay5 THEN
		step := 6;
		last := tx;
	END_IF;
END_IF;
IF run AND step = 6 THEN
	IF NOT q6 AND in6 AND tx - last <= wait6 THEN
		Q5 := FALSE;
		Q6 := TRUE;
		last := tx;
	ELSIF NOT q6 AND Tx - last > wait6 THEN
		status := 7;
		q5 := FALSE;
		run := FALSE;
	ELSIF q6 AND tx - last >= delay6 THEN
		step := 7;
		last := tx;
	END_IF;
END_IF;
IF run AND step = 7 THEN
	IF NOT q7 AND in7 AND tx - last <= wait7 THEN
		Q6 := FALSE;
		Q7 := TRUE;
		last := tx;
	ELSIF NOT q7 AND Tx - last > wait7 THEN
		status := 8;
		q6 := FALSE;
		run := FALSE;
	ELSIF q7 AND tx - last >= delay7 THEN
		step := -1;
		Q7 := FALSE;
		Run := FALSE;
		status := 110;
	END_IF;
END_IF;
any := q0 OR q1 OR q2 OR q3 OR q4 OR q5 OR q6 OR q7;

(*
hm 1.10.06		rev 1.1
	corrected delay logic to be after event and not before
	added any output

hm 1.12.06		rev 1.2
	corrected failure in sequence logic.
	added init at startup to prevent from initial statuss after start.

hm 17.1.2007		rev 1.3
	changed output fault to status for better compatibility with other modules (ESR)
	added stop on error functionality and setup variable
	default for inputs in0..7 is true.
	renames variable state to step

hm	17.sep 2007		rev 1.4
	replaced time() with T_PLC_MS() for compatibility reasons

*)
END_FUNCTION_BLOCK

(* POU Engineering/control/hyst_1, ST *)
FUNCTION_BLOCK hyst_1
VAR_INPUT
	In : REAL;
	high : REAL;
	low : REAL;
END_VAR
VAR_OUTPUT
	Q : BOOL := 0;
	win : BOOL := 0;
END_VAR
VAR
END_VAR

(*
	version 1.0	4 aug 2006
	programmer 	hugo
	tested BY		tobias

this hysteresis function switches the output high if the input signal reaches obove high and will switch to low when the input falls back below low value.
a separate output mid is set if the input stays between low and high value.

*)
IF Q THEN
	IF in < low THEN q := FALSE; END_IF;
ELSE
	IF in > high THEN q := TRUE; END_IF;
END_IF;
win := in > low AND in < high;
END_FUNCTION_BLOCK

(* POU Building/HLK/temp_ext, ST *)
FUNCTION_BLOCK temp_ext
VAR_INPUT
	t_ext1 : REAL;
	t_ext2 : REAL;
	t_ext3 : REAL;
	t_ext_config : BYTE := 0;
	dt_in : DT;
END_VAR
VAR_INPUT CONSTANT
	t_ext_min : REAL := -40;
	t_ext_max : REAL := 60;
	t_ext_default : REAL := -10;
	heat_period_start : DATE := D#1970-9-1;
	heat_period_stop : DATE := D#1970-4-30;
	cool_period_start : DATE := D#1970-4-1;
	cool_period_stop : DATE := D#1970-9-30;
	heat_start_temp_day : REAL := 15;
	heat_start_temp_night : REAL := 10;
	heat_stop_temp : REAL := 18;
	cool_start_temp_day : REAL := 26;
	cool_start_temp_night : REAL := 26;
	cool_stop_temp : REAL := 24;
	start_day : TOD := tod#09:00;
	start_night : TOD := tod#21:00;
	cycle_time : TIME := t#10m;
END_VAR
VAR_OUTPUT
	t_ext : REAL;
	heat : BOOL;
	cool : BOOL;
END_VAR
VAR
	tx: TIME;
	last_run: TIME;
	init: BOOL;
	cool_start: DATE;
	cool_stop: DATE;
	heat_start: DATE;
	heat_stop: DATE;
	xdate: DATE;
	day: BOOL;
END_VAR


(*
version 1.1	15 sep 2007
programmer 	hugo
tested by		tobias

temp_ext measures and processes ext temperature and decides if heating or cooling is needed.

 the measurement of t_ext has 3 inputs which can be configured in different ways:
	t_ext_config = 0 means the ext temp is the avg of the 3 external temperatures, this mode is the default mode.
	t_ext_config = 1 means t_ext1 is used.
	t_ext_config = 2 means t_ext1 is used.
	t_ext_config = 3 means t_ext1 is used.
	t_ext_config = 4 means t_ext_default is used.
	t_ext_config = 5 means the lowest of the 3 external temperatures is used.
	t_ext_config = 6 means the higest externnal temperature is used.
	t_ext_config = 7 means the midlle external temperature is used, if there are only two working, the lowest is used.
	in any config mode, an external temperature higher then t_ext_max or lower then t_ext_min is ignored to prevent from temperatures caused by broken sensors or wires.
	if no external temperature is available, a default value (t_ext_default) is used.
	if you have only one external sensor, connect the 3 inputs to the same sensor, or select the right input with t_ext_config.

heating or cooling is enabled during heating / cooling period when the day or night start temperature is reached for at least the specified delay time and will be disabled after the stop temperature is reached. 
t_ext output can be used by other modules to determine the correct system temperature for heating or cooling.

*)
IF NOT init THEN
	init := TRUE;
	heat_start := set_Date(1972,month(heat_period_start),day_of_month(heat_period_start));
	heat_stop := set_Date(1972,month(heat_period_stop),day_of_month(heat_period_stop));
	cool_start := set_Date(1972,month(cool_period_start),day_of_month(cool_period_start));
	cool_stop := set_Date(1972,month(cool_period_stop),day_of_month(cool_period_stop));
END_IF;

(* read system time *)
tx := DWORD_TO_TIME(T_PLC_MS());

(* for efficiency exit isf this program has been executed less then 1min ago *)
IF tx - last_run < cycle_time THEN RETURN; END_IF;

(* calculate frequently used variables *)
xdate := set_Date(1972,month(DT_TO_DATE(dt_in)),day_of_month(DT_TO_DATE(dt_in)));
day := DT_TO_TOD(dt_in) >= start_day AND  DT_TO_TOD(dt_in) < start_night;

(* read the correct external temperature depending on the t_ext_config setting *)
t_ext := multi_in(t_ext1, t_ext2, t_ext3, t_ext_default, t_ext_min, t_ext_max, t_ext_config);

(* dtermine heating *)
IF (heat_start <= heat_stop AND xdate >= heat_start AND xdate <= heat_stop) OR (heat_start > heat_stop AND (xdate >= heat_start OR xdate <= heat_stop)) THEN
	(* heating period id true check for temperature *)
	IF day AND t_ext <= heat_start_temp_day THEN
		heat := TRUE;
	ELSIF NOT day AND t_ext <= heat_start_temp_night THEN
		heat := TRUE;
	ELSIF t_ext >= heat_stop_temp THEN
		heat := FALSE;
	END_IF;
ELSE
	heat := FALSE;
END_IF;

(* dtermine cooling *)
IF (cool_start <= cool_stop AND xdate >= cool_start AND xdate <= cool_stop) OR (cool_start > cool_stop AND (xdate >= cool_start OR xdate <= cool_stop)) THEN
	(* cooling period is true check for temperature *)
	IF day AND t_ext >= cool_start_temp_day THEN
		cool := TRUE;
	ELSIF NOT day AND t_ext >= cool_start_temp_night THEN
		cool := TRUE;
	ELSIF t_ext <= cool_stop_temp THEN
		cool := FALSE;
	END_IF;
ELSE
	cool := FALSE;
END_IF;

last_run := tx;

(* revision history
hm	6 dec 2006		rev 1.0
	original version

hm	15.9.2007		rev 1.1
	replaced Time() with T_PLC_MS for compatibility and performance reasons

*)
END_FUNCTION_BLOCK

(* POU Engineering/sensor/multi_in, ST *)
FUNCTION multi_in : REAL
VAR_INPUT
	in_1 : REAL;
	in_2 : REAL;
	in_3 : REAL;
	default : REAL;
	in_min : REAL;
	in_max : REAL;
	mode : BYTE;
END_VAR
VAR
	count: INT;
	F1: BOOL;
	F2: BOOL;
	F3: BOOL;
END_VAR

(*

version 1.1	1 jan 2007
programmer 	oscat
tested by		hugo

multi_in is a signal conditioning function ehich can be configured in 8 different ways.
it is used to read multiple sensors for the same value and protect the user from broken sensors or invalid data from sensors.

multi_in can be configured in different ways:
	mode = 0 means the the avg of the 3 inputs is used, this mode is the default mode.
	mode = 1 means in_1 is used.
	mode = 2 means in_2 is used.
	mode = 3 means in_3 is used.
	mode = 4 means default is used.
	mode = 5 means the lowest of the 3 external temperatures is used.
	mode = 6 means the higest externnal temperature is used.
	mode = 7 means the midlle input is used, if there are only two working, the lowest input is used.
	mode > 7 ,eans output is 0 at all times.
	in any config mode, an input higher then in_max or lower then in_min is ignored to prevent values from broken sensors or wires.
	if all inputs are higher then in_max or lower then in_min, a default value (default) is used.
*)
IF  in_1 > in_min AND in_1 < in_max THEN F1 := TRUE; ELSE F1 := FALSE; END_IF;
IF  in_2 > in_min AND in_2 < in_max THEN F2 := TRUE; ELSE F2 := FALSE; END_IF;
IF  in_2 > in_min AND in_3 < in_max THEN F3 := TRUE; ELSE F3 := FALSE; END_IF;

CASE mode OF
0:	count := 0;
	IF F1 THEN
		count := count + 1;
		multi_in := in_1;
	ELSE
		multi_in := 0;
	END_IF;
	IF F2 THEN
		count := count + 1;
		multi_in := multi_in + in_2;
	END_IF;
	IF F3 THEN
		count := count + 1;
		multi_in := multi_in + in_3;
	END_IF;
	IF count = 0 THEN
		multi_in := default;
	ELSE
		multi_in := multi_in / count;
	END_IF;

1:	IF F1 THEN multi_in := in_1; ELSE multi_in := default; END_IF;

2:	IF F2 THEN multi_in := in_2; ELSE multi_in := default; END_IF;

3:	IF F3 THEN multi_in := in_3; ELSE multi_in := default; END_IF;

4:	multi_in := default;

5:	IF F1 THEN multi_in := in_1; ELSE multi_in := in_max; END_IF;
	IF F2 AND in_2 < multi_in THEN multi_in := in_2; END_IF;
	IF F3 AND in_3 < multi_in THEN multi_in := in_3; END_IF;
	IF multi_in = in_max THEN multi_in := default; END_IF;

6:	IF F1 THEN multi_in := in_1; ELSE multi_in := in_min; END_IF;
	IF F2 AND in_2 > multi_in THEN multi_in := in_2; END_IF;
	IF F3 AND in_3 > multi_in THEN multi_in := in_3; END_IF;
	IF multi_in = in_min THEN multi_in := default; END_IF;

7:	IF F1 AND F2 AND F3 THEN multi_in := mid3(in_1, in_2, in_3);
	ELSIF F1 AND F2 THEN multi_in := MIN(in_1, in_2);
	ELSIF F1 AND F3 THEN multi_in := MIN(in_1, in_3);
	ELSIF F2 AND F3 THEN multi_in := MIN(in_2, in_3);
	ELSIF F1 THEN multi_in := in_1;
	ELSIF F2 THEN multi_in := in_2;
	ELSIF F3 THEN multi_in := in_3;
	ELSE multi_in := default;
	END_IF;

END_CASE;

(*
hm 1.1.2007	rev 1.1
	changed midr to mid3 function

*)
END_FUNCTION

(* POU Engineering/automation/FT_Profile, ST *)
FUNCTION_BLOCK FT_Profile
VAR_INPUT
	K : REAL := 1;
	O : REAL := 0;
	M : REAL := 1;
	E : BOOL;
END_VAR
VAR_INPUT CONSTANT
	value_0 : REAL;
	time_1 : TIME;
	value_1 : REAL;
	time_2 : TIME;
	value_2 : REAL;
	time_3 : TIME;
	value_3 : REAL;
	time_10 : TIME;
	value_10 : REAL;
	time_11 : TIME;
	value_11 : REAL;
	time_12 : TIME;
	value_12 : REAL;
	time_13 : TIME;
	value_13 : REAL;
END_VAR
VAR_OUTPUT
	Y : REAL;
	RUN : BOOL;
	ET : TIME;
END_VAR
VAR
	tx : TIME;
	edge : BOOL;
	state: BYTE;
	ta: TIME;
	tb: TIME;
	t0 : TIME;
	temp: REAL;
	va: REAL;
	vb: REAL;
END_VAR

(*
version 1.1	15 sep 2007
programmer 	tobias
tested by		hugo

FT_Profile generates an output signal which is defined by values over a time scale.
the different values are connected by ramps between the individual values.
a rising edge on E starts the output signal generation and E = True can delay time_3 / value_3 as long as it stays true.
an additional multiplier K can be used to multiply the output and an offset O can be added to the output dynamically.
*)
(* read system time *)
tx := DWORD_TO_TIME(T_PLC_MS());

(* determine start condition *)
IF E AND NOT edge THEN
	RUN := TRUE;
	ET := t#0s;
	t0 := tx;
	ta := tx;
	tb := multime(time_1, M);
	va := value_0;
	vb := value_1;
	temp := value_0;
	state := 1;
END_IF;
edge := E;

(* generate startup profile *)
IF run THEN
	CASE state OF
		1:	IF tx - ta >= tb THEN
				ta := ta + tb;
				tb := multime(time_2 - time_1, M);
				va := value_1;
				vb := value_2;
				temp := value_1;
				state := 2;
			ELSE
				temp := ((vb - va) * TIME_TO_REAL(tx - ta) / TIME_TO_REAL(tb) + va);
			END_IF;
		2:	IF tx - ta >= tb THEN
				ta := ta + tb;
				tb := multime(time_3 - time_2, M);
				va := value_2;
				vb := value_3;
				temp := value_2;
				state := 3;
			ELSE
				temp := ((vb - va) * TIME_TO_REAL(tx - ta) / TIME_TO_REAL(tb) + va);
			END_IF;
		3:	IF tx - ta >= tb THEN
				ta := ta + tb;
				tb := multime(time_10 - time_3, M);
				va := value_3;
				vb := value_10;
				temp := value_3;
				state := 4;
			ELSE
				temp := ((vb - va) * TIME_TO_REAL(tx - ta) / TIME_TO_REAL(tb) + va);
			END_IF;
		4 :	IF tx - ta >= tb THEN
				ta := ta + tb;
				tb := multime(time_11 - time_10, M);
				va := value_10;
				vb := value_11;
				temp := value_10;
				IF E THEN state := 5; ELSE state := 6; END_IF;
			ELSE
				temp := ((vb - va) * TIME_TO_REAL(tx - ta) / TIME_TO_REAL(tb) + va);
			END_IF;
		5:	(* extend the signal while E is true *)
			IF E THEN
				ta := tx;
			ELSE
				state := 6;
			END_IF;
		6:	IF tx - ta >= tb THEN
				ta := ta + tb;
				tb := multime(time_12 - time_11, M);
				va := value_11;
				vb := value_12;
				temp := value_11;
				state := 7;
			ELSE
				temp := ((vb - va) * TIME_TO_REAL(tx - ta) / TIME_TO_REAL(tb) + va);
			END_IF;
		7:	IF tx - ta >= tb THEN
				ta := ta + tb;
				tb := multime(time_13 - time_12, M);
				va := value_12;
				vb := value_13;
				temp := value_12;
				state := 8;
			ELSE
				temp := ((vb - va) * TIME_TO_REAL(tx - ta) / TIME_TO_REAL(tb) + va);
			END_IF;
		8:	IF tx - ta >= tb THEN
				temp := value_13;
				run := FALSE;
			ELSE
				temp := ((vb - va) * TIME_TO_REAL(tx - ta) / TIME_TO_REAL(tb) + va);
			END_IF;
	END_CASE;
	Y := temp * K + O;
	ET := tx - t0;
END_IF;

(* revision history
hm	27 feb 2007		rev 1.0
	original version

hm	15. sep2007		rev 1.1
	replaced Time() with T_PLC_MS for compatibility and performance reasons

*)
END_FUNCTION_BLOCK

(* POU Engineering/control/FT_IMP, ST *)
FUNCTION_BLOCK FT_IMP
VAR_INPUT
	in : REAL;
	T : TIME;
	K : REAL := 1;
END_VAR
VAR_OUTPUT
	out : REAL;
END_VAR
VAR
	t1 : FT_PT1;
END_VAR

(*
version 1.1	3 Jan 2007
programmer 	hugo
tested by		tobias

FT_IMP is 	an impulse filter (high pass filter) with the time T and factor K.
 
*)
T1(in:= in, T:=T);
out := (in - t1.out) * K;

(*
hm 3.1.2007	rev 1.1
	added factor K

*)
END_FUNCTION_BLOCK

(* POU Engineering/control/FT_TN16, ST *)
FUNCTION_BLOCK FT_TN16
VAR_INPUT
	in : REAL;
	T : TIME;
END_VAR
VAR_OUTPUT
	out : REAL;
	trig : BOOL;
END_VAR
VAR
	length : INT := 16;
	X : ARRAY[0..15] OF REAL;
	cnt : INT;
	last : TIME;
	tx: TIME;
	init: BOOL;
END_VAR

(*
version 1.1	16 sep 2007
programmer 	hugo
tested by		tobias

FT_TN16 is delay function, it will delay a signal by a specified time : T and will store 16 values of in before they are put thru to out.
for higher or lower resolution please use FT_TN8 or FT_TN64 instead.
 
*)
(* read system time *)
tx := DWORD_TO_TIME(T_PLC_MS());

trig := FALSE;
IF NOT init THEN
	x[cnt] := in;
	init := TRUE;
	last := tx;
ELSIF tx - last >= T / length THEN
	IF cnt = length - 1 THEN cnt := 0; ELSE cnt := cnt + 1; END_IF;
	Out := X[cnt];
	x[cnt] := in;
	last := tx;
	Trig := TRUE;
END_IF;

(* revision history
hm		1. jan 2007		rev 1.0
	original version

hm		16. sep 2007	rev 1.1
	changes time() to T_plc_ms() for compatibility reasons

*)
END_FUNCTION_BLOCK

